TYPE UDT 31
VERSION : 0.0
  STRUCT
   A_FD_OR : BYTE ;	//Feedrate override
   A_DriveEnable : BOOL ;	//Drive test movement enable
   A_AckFixedStop : BOOL ;	//Acknowledge fixed stop reached
   A_SensorFixedStop : BOOL ;	//Sensor fixed stop
   A_ASpDisable : BOOL ;	//Axis/spindle disable
   A_Follow_upMode : BOOL ;	//Follow-up mode
   A_PosMeas1 : BOOL ;	//Position measuring system 1
   A_PosMeas2 : BOOL ;	//Position measuring system 2
   A_ORactive : BOOL ;	//Override active
   A_SWCam : BOOL ;	//SW cam activation
   A_ContrEnable : BOOL ;	//Controller enable
   A_DelDTGSpReset : BOOL ;	//Delete distance to go/Spindle-Reset
   A_Clamp : BOOL ;	//Clamping in progress
   A_RefVal1 : BOOL ;	//Reference point value 1
   A_RefVal2 : BOOL ;	//Reference point value 2
   A_RefVal3 : BOOL ;	//Reference point value 3
   A_RefVal4 : BOOL ;	//Reference point value 4
   A_ExtZO : BOOL ;	//Import external ZO
   A_EnabTravFixedStop : BOOL ;	//Enable travel to fixed stop
   A_FixedFD1 : BOOL ;	//Activate fixed feed 1
   A_FixedFD2 : BOOL ;	//Activate fixed feed 2
   A_FixedFD3 : BOOL ;	//Activate fixed feed 3
   A_FixedFD4 : BOOL ;	//Activate fixed feed 4
   A_VelocSpeedLimit : BOOL ;	//Velocity/spindle speed limitation
   A_PrgtestAxRel : BOOL ;	// Program test axis/spindle release
   A_HW1 : BOOL ;	//Activate handwheel 1
   A_HW2 : BOOL ;	//Activate handwheel 2
   A_HW3 : BOOL ;	//Activate handwheel 3
   A_FDSpStop : BOOL ;	//Feed stop/spindle stop
   A_Disable : BOOL ;	//Traversing key disable
   A_RapidTrOR : BOOL ;	//Rapid traverse override
   A_Minus : BOOL ;	//Traversing key minus
   A_Plus : BOOL ;	//Traversing key plus
   A_INC1 : BOOL ;	//INC1
   A_INC10 : BOOL ;	//INC10
   A_INC100 : BOOL ;	//INC100
   A_INC1000 : BOOL ;	//INC1000
   A_INC10000 : BOOL ;	//INC10000
   A_INCVar : BOOL ;	//INC variable
   A_OEMAxis : BYTE ;	//OEM axis signals
   f7 : BYTE ;
   A_NCASpChanA : BOOL ;	//Assign NC axis/spindle channel A
   A_NCASpChanB : BOOL ;	//Assign NC axis/spindle channel B
   A_NCASpChanC : BOOL ;	//Assign NC axis/spindle channel C
   A_NCASpChanD : BOOL ;	//Assign NC axis/spindle channel D
   A_NCASpStrobe : BOOL ;	//Activation of assignment with pos. edge
   f8_5 : BOOL ;
   f8_6 : BOOL ;
   A_PLCASp : BOOL ;	//Request PLC axis/spindle
   A_Para_A : BOOL ;	//Parameter block servo A
   A_Para_B : BOOL ;	//Parameter block servo B
   A_Para_C : BOOL ;	//Parameter block servo C
   A_LockParSetDef : BOOL ;	//Lock parameter set definition from NC
   f9_4 : BOOL ;
   f9_5 : BOOL ;
   f9_6 : BOOL ;
   f9_7 : BOOL ;
   A_REPOSDelay : BOOL ;	//REPOS DELAY
   f10_1 : BOOL ;
   f10_2 : BOOL ;
   f10_3 : BOOL ;
   f10_4 : BOOL ;
   f10_5 : BOOL ;
   f10_6 : BOOL ;
   f10_7 : BOOL ;
   A_StartBrakeTest : BOOL ;	// Start brake test
   f11_1 : BOOL ;
   f11_2 : BOOL ;
   f11_3 : BOOL ;
   f11_4 : BOOL ;
   f11_5 : BOOL ;
   f11_6 : BOOL ;
   f11_7 : BOOL ;
   A_HWLimitMinus : BOOL ;	//Hardware limit switch minus
   A_HWLimitPlus : BOOL ;	//Hardware limit switch plus
   A_SWLimit2Minus : BOOL ;	//2nd software limit switch minus
   A_SWLimit2Plus : BOOL ;	//2nd software limit switch plus
   A_ModuloLimitEn : BOOL ;	// Modulo limit enabled
   f12_5 : BOOL ;
   f12_6 : BOOL ;
   A_DelayRef : BOOL ;	//Delay reference point approach
   f13 : BYTE ;
   f14 : INT ;
   A_ActGearA : BOOL ;	//Actual gear stage A
   A_ActGearB : BOOL ;	//Actual gear stage B
   A_ActGearC : BOOL ;	//Actual gear stage C
   A_GearChangeOv : BOOL ;	//Gear has changed over
   A_Sp1Syn : BOOL ;	//Re-synchronize spindle 1
   A_Sp2Syn : BOOL ;	//Re-synchronize spindle 2
   A_NoMonitorGear : BOOL ;	//No monitoring when changing gear
   A_DeleteS : BOOL ;	//Delete S value
   A_FD_ORSp : BOOL ;	//Feedrate override for spindle valid
   f17_1 : BOOL ;
   f17_2 : BOOL ;
   f17_3 : BOOL ;
   A_Sp1SynP : BOOL ;	//Re-synchronize spindle 1 f. positioning
   A_Sp2SynP : BOOL ;	//Re-synchronize spindle 2 f. positioning
   A_M3M4Inv : BOOL ;	//Invert M3/M4
   f17_7 : BOOL ;
   f18_0 : BOOL ;
   f18_1 : BOOL ;
   f18_2 : BOOL ;
   f18_3 : BOOL ;
   A_OscilPLC : BOOL ;	//Oscillation via PLC
   A_OscilSpeed : BOOL ;	//enable Oscillation
   A_SetRotDirectRight : BOOL ;	//Setpoint osci. direct. right
   A_SetRotDirectLeft : BOOL ;	//Setpoint osci. direct. left
   A_SpOR : BYTE ;	//Spindle override
   A_UFSwOv : BOOL ;	//Run-up switchover U/F operation
   A_RUEncQuStop : BOOL ;	//Run-up encoder quick stop
   A_Tlimit2 : BOOL ;	//Torque limit 2
   A_SpeedSetpSmooth : BOOL ;	//Speed setpoint smoothing
   f20_4 : BOOL ;
   A_HoldBrakeToOpen : BOOL ;	// holding brake open
   f20_6 : BOOL ;
   f20_7 : BOOL ;
   A_ParA : BOOL ;	//Parameter set selection A
   A_ParB : BOOL ;	//Parameter set selection B
   A_ParC : BOOL ;	//Parameter set selection C
   A_MotA : BOOL ;	//Motor selection A
   A_MotB : BOOL ;	//Motor selection B
   A_MotOK : BOOL ;	//Motor selected
   A_IntegratDisable : BOOL ;	//n controller integrator disable
   A_PulseEnable : BOOL ;	//Pulse enable
   A_SG_SBH : BOOL ;	//Deselection SG/SBH
   A_SBH : BOOL ;	//Deselection of safe standstill
   f22_2 : BOOL ;
   A_SGselect0 : BOOL ;	//Selection SG bit 0
   A_SGselect1 : BOOL ;	//Selection SG bit 1
   f22_5 : BOOL ;
   f22_6 : BOOL ;
   f22_7 : BOOL ;
   A_Transmiss0 : BOOL ;	//Selection Transmission bit 0
   A_Transmiss1 : BOOL ;	//Selection Transmission bit 1
   A_Transmiss2 : BOOL ;	//Selection Transmission bit 2
   f23_3 : BOOL ;
   A_SE : BOOL ;	//Selection SE
   A_BrakeToClose : BOOL ;	// Sinamics: Brake to close
   f23_6 : BOOL ;
   A_TestStop : BOOL ;	//Activate test stop
   A_RotationMonit : BOOL ;	// Stepper motor: Rotation monitoring
   A_ControlAx : BOOL ;	// Control Axis
   f24_2 : BOOL ;
   f24_3 : BOOL ;
   A_TorqComp : BOOL ;	// Torque compensation
   A_ChangSetpOutAss0 : BOOL ;	// Bit value for CTRLOUT_changed - Change setpoint output assignment
   A_ChangSetpOutAss1 : BOOL ;	// Bit value for CTRLOUT_changed - Change setpoint output assignment
   A_MS : BOOL ;	//Master / Slave On
   f25 : BYTE ;
   f26_0 : BOOL ;
   f26_1 : BOOL ;
   f26_2 : BOOL ;
   A_CompContr : BOOL ;	//Compensation controller On
   A_FollowAxOv : BOOL ;	//Enable following axis override
   f26_5 : BOOL ;
   f26_6 : BOOL ;
   f26_7 : BOOL ;
   A_DEPMCS : BOOL ;	// Resume: DEPMCS
   A_DEPBCS : BOOL ;	// Resume: DEPBCS
   A_Corr : BOOL ;	// Resume: Corr
   A_HIAxMove : BOOL ;	// Resume: HIAxMove
   A_StopDEPMCS : BOOL ;	// Stop: DEPMCS
   A_StopDEPBCS : BOOL ;	// Stop: DEPBCS
   A_StopCorr : BOOL ;	// Stop: Corr
   A_StopHIAxMove : BOOL ;	// Stop: HIAxMove
   A_OscillAxExtRev : BOOL ;	// OscillAxExtReversal
   A_AxReset : BOOL ;	// AXRESET
   A_AxResume : BOOL ;	// AXRESUME
   A_SetRP : BOOL ;	//Set reversal point
   A_ChangeRP : BOOL ;	//Change reversal point
   A_StopRP : BOOL ;	//Stop at next reversal point
   A_Stop : BOOL ;	//Stop
   A_PLCAxis : BOOL ;	//PLC checks axis
   f29_0 : BOOL ;
   f29_1 : BOOL ;
   f29_2 : BOOL ;
   f29_3 : BOOL ;
   A_StartGantSynRun : BOOL ;	//Start gantry synchronization run
   A_NoAutoSync : BOOL ;	//No auto sync
   f29_6 : BOOL ;
   f29_7 : BOOL ;
   A_StopSpindle : BOOL ;	//Stop spindle
   A_StartCW : BOOL ;	//Start spindle Clockwise
   A_StartCCW : BOOL ;	//Start spindle Counterclockwise
   A_AutoGearStep : BOOL ;	//Autom. gear step change
   A_PosSpindle : BOOL ;	//Position spindle
   f30_5 : BOOL ;
   f30_6 : BOOL ;
   f30_7 : BOOL ;
   f31_0 : BOOL ;
   f31_1 : BOOL ;
   f31_2 : BOOL ;
   f31_3 : BOOL ;
   A_Resynchronize : BOOL ;	// Resynchronize
   A_DisSync : BOOL ;	// Disable synchronization
   A_Tracksync : BOOL ;	// Track synchronism
   f31_7 : BOOL ;
   f32_0 : BOOL ;
   f32_1 : BOOL ;
   A_extStopA : BOOL ;	//Deselection external Stop A
   A_extStopC : BOOL ;	//Deselection external Stop C
   A_extStopD : BOOL ;	//Deselection external Stop D
   A_extStopE : BOOL ;	//Deselection external Stop E
   f32_6 : BOOL ;
   f32_7 : BOOL ;
   f33_0 : BOOL ;
   f33_1 : BOOL ;
   f33_2 : BOOL ;
   f33_3 : BOOL ;
   A_SGcorr_0 : BOOL ;	//Selection SG-correction Bit 0
   A_SGcorr_1 : BOOL ;	//Selection SG-correction Bit 1
   A_SGcorr_2 : BOOL ;	//Selection SG-correction Bit 2
   A_SGcorr_3 : BOOL ;	//Selection SG-correction Bit 3
   f34 : ARRAY  [34 .. 55 ] OF BYTE ;
   A_FeedDriveCAxEng : BOOL ;	// Seperate feed drive as C axis engaged
   A_SpSpeedDisp : BOOL ;	// Spindle speed display
   A_SpInsideClamp : BOOL ;	// Spindle inside clamping
   f56_3 : BOOL ;
   f56_4 : BOOL ;
   f56_5 : BOOL ;
   f56_6 : BOOL ;
   f56_7 : BOOL ;
   f57 : BYTE ;
   f58 : WORD ;	// FC18: internal
   E_SpNA : BOOL ;	//Spindle/no axis
   E_NCU_Link : BOOL ;	//NCU_link active axis
   E_EncodFreq1 : BOOL ;	//Encoder limit frequency 1 exceeded
   E_EncodFreq2 : BOOL ;	//Encoder limit frequency 2 exceeded
   E_RefSyn1 : BOOL ;	//Referenced/synchronized 1
   E_RefSyn2 : BOOL ;	//Referenced/synchronized 2
   E_ExactCoarse : BOOL ;	//Position reached with exact stop coarse
   E_ExactFine : BOOL ;	//Position reached with exact stop fine
   E_TravRequ : BOOL ;	//Travel request
   E_AxialAlarm : BOOL ;	// Axial alarm
   E_AxisReady : BOOL ;	//Axis ready
   E_Follow_upMode : BOOL ;	//Follow-up mode active
   E_Stat : BOOL ;	//Axis/spindle stationary (n<nmin)
   E_PositContr : BOOL ;	//Position controller active
   E_SpeedContr : BOOL ;	//Speed controller active
   E_CurrentContr : BOOL ;	//Current controller active
   E_SWCam : BOOL ;	//Software cams active
   E_HWOverlay : BOOL ;	//Handwheel overlay active
   E_RevFD : BOOL ;	//Revolutional feedrate active
   E_MeasAct : BOOL ;	//Measuring active
   E_ActTravFStop : BOOL ;	//Activate travel to fixed stop
   E_FixedStop : BOOL ;	//Fixed stop reached
   E_ForceFixedStop : BOOL ;	// Force fixed stop limited
   E_AxContainerRot : BOOL ;	// Axis container rotation active
   E_AxReset : BOOL ;	// Axis reset done
   E_PLCCtrlAx : BOOL ;	// PLCcontrolled axis
   E_AxStop : BOOL ;	// Axis stop active
   E_AxSpDisable : BOOL ;	// Axis/spindle disable active
   E_StopDEPMCS : BOOL ;	// stop DEPMCS active
   E_StopDEPBCS : BOOL ;	// stop DEPBCS active
   E_StopCorr : BOOL ;	// stop Corr active
   E_StopHIAxMove : BOOL ;	// Stop HIAxMove active
   E_HW1 : BOOL ;	//Handwheel 1 active
   E_HW2 : BOOL ;	//Handwheel 2 active
   E_HW3 : BOOL ;	//Handwheel 3 active
   f64_3 : BOOL ;
   E_TReqMinus : BOOL ;	// Travel request minus
   E_TReqPlus : BOOL ;	// Travel request plus
   E_TCMinus : BOOL ;	//Traverse command minus
   E_TCPlus : BOOL ;	//Traverse command plus
   E_INC1 : BOOL ;	//INC1
   E_INC10 : BOOL ;	//INC10
   E_INC100 : BOOL ;	//INC100
   E_INC1000 : BOOL ;	//INC1000
   E_INC10000 : BOOL ;	//INC10000
   E_INCVar : BOOL ;	//INC variable
   f65_6 : BOOL ;
   f65_7 : BOOL ;
   E_OEMAxis : BYTE ;	//OEM axis signals
   f67 : BYTE ;
   E_NCASpChanA : BOOL ;	//NC axis/spindle in channel A
   E_NCASpChanB : BOOL ;	//NC axis/spindle in channel B
   E_NCASpChanC : BOOL ;	//NC axis/spindle in channel C
   E_NCASpChanD : BOOL ;	//NC axis/spindle in channel D
   E_PLCType : BOOL ;	//New type requested by PLC
   E_ChPoss : BOOL ;	//Change axis possible
   E_NeutrASp : BOOL ;	//Neutral axis/spindle
   E_PLCASp : BOOL ;	//PLC axis/spindle
   E_ParS_A : BOOL ;	//Parameter block servo A
   E_ParS_B : BOOL ;	//Parameter block servo B
   E_ParS_C : BOOL ;	//Parameter block servo C
   E_ReposSh : BOOL ;	// Repos shift
   E_ReposShValid : BOOL ;	// Repos shift valid
   E_ReposDelayQuit : BOOL ;	// Repos delay quit
   f70_3 : BOOL ;
   f70_4 : BOOL ;
   f70_5 : BOOL ;
   f70_6 : BOOL ;
   f70_7 : BOOL ;
   E_BrakeTest : BOOL ;	// Brake test active
   f71_1 : BOOL ;
   f71_2 : BOOL ;
   f71_3 : BOOL ;
   f71_4 : BOOL ;
   f71_5 : BOOL ;
   f71_6 : BOOL ;
   E_PLCAxDedic : BOOL ;	// PLC Axis dedicated
   E_MMC_REPOSDelay : BOOL ;	//MMC REPOS DELAY
   f72_1 : BOOL ;
   f72_2 : BOOL ;
   f72_3 : BOOL ;
   f72_4 : BOOL ;
   f72_5 : BOOL ;
   f72_6 : BOOL ;
   f72_7 : BOOL ;
   f73 : BYTE ;
   f74_0 : BOOL ;
   f74_1 : BOOL ;
   f74_2 : BOOL ;
   f74_3 : BOOL ;
   E_ModLimEnAct : BOOL ;	// Modulo limit enabled active
   f74_5 : BOOL ;
   f74_6 : BOOL ;
   f74_7 : BOOL ;
   f75 : BYTE ;
   E_ScratchPulse : BOOL ;	//Scratch pulse
   f76_1 : BOOL ;
   f76_2 : BOOL ;
   f76_3 : BOOL ;
   E_PathAxis : BOOL ;	// Path axis
   E_PosAxis : BOOL ;	//Positioning axis
   E_IndexAxisPos : BOOL ;	//Indexing axis in position
   E_CurvePos : BOOL ;	//Curve axis in position
   E_CollCheckRedSpeed : BOOL ;	//reduced speed of Collisions Check
   f77_1 : BOOL ;
   f77_2 : BOOL ;
   f77_3 : BOOL ;
   f77_4 : BOOL ;
   f77_5 : BOOL ;
   f77_6 : BOOL ;
   f77_7 : BOOL ;
   E_FPosAxis : REAL ;	//F function (REAL format) for positioning axes
   E_SetpGearA : BOOL ;	//Setpoint gear stage A
   E_SetpGearB : BOOL ;	//Setpoint gear stage B
   E_SetpGearC : BOOL ;	//Setpoint gear stage C
   E_GearChange : BOOL ;	//Gear changeover
   f82_4 : BOOL ;
   f82_5 : BOOL ;
   f82_6 : BOOL ;
   f82_7 : BOOL ;
   E_SpeedLimit : BOOL ;	//Speed limit exceeded
   E_SetSpeedLimit : BOOL ;	//Setpoint speed limited
   E_SetSpeedIncreased : BOOL ;	//Setpoint speed increased
   E_GeoMonit : BOOL ;	//Geometry monitoring
   E_SupportAreaViol : BOOL ;	//Support area limits violated
   E_SetRange : BOOL ;	//Spindle in setpoint range
   E_SpeedMonit : BOOL ;	//Speed monitoring
   E_ActRotRight : BOOL ;	//Actual rotation direction right
   E_ConstCuttSpeed : BOOL ;	//Const. cutting speed active
   E_SUG : BOOL ;	//SUG active (grinding wheel surface speed)
   E_CLG : BOOL ;	//CLG active
   E_Tapping : BOOL ;	//Tapping without compensating chuck
   E_SyncMode : BOOL ;	//Synchronous mode spindle active
   E_PosMode : BOOL ;	//Positioning mode spindle active
   E_OscillMode : BOOL ;	//Oscillation mode spindle active
   E_ContrMode : BOOL ;	//Control mode spindle active
   f85_0 : BOOL ;
   f85_1 : BOOL ;
   f85_2 : BOOL ;
   f85_3 : BOOL ;
   f85_4 : BOOL ;
   E_SpInPosition : BOOL ;	// Spindle in position
   f85_6 : BOOL ;
   f85_7 : BOOL ;
   E_MFunct : INT ;	//M function (INT) for spindle
   E_SFunct : REAL ;	//S function (REAL) for spindle
   E_SetUpMode : BOOL ;	//Set-up mode active
   E_RUEncDisabl : BOOL ;	//Run-up encoder disable active
   E_Tlimit2 : BOOL ;	//Torque limit 2 active
   E_SpeedSetpSmooth : BOOL ;	//Speed setpoint smoothing active
   E_RLIact : BOOL ;	// RLI active
   E_HoldBrakeOpened : BOOL ;	// holding brake opened
   E_EarthFaultDetec : BOOL ;	// earth-fault detection
   f92_7 : BOOL ;
   E_ParA : BOOL ;	//Active parameter set A
   E_ParB : BOOL ;	//Active parameter set B
   E_ParC : BOOL ;	//Active parameter set C
   E_MotA : BOOL ;	//Active motor A
   E_MotB : BOOL ;	//Active motor B
   E_MotOK : BOOL ;	//Drive ready
   E_IntegratDisable : BOOL ;	//n controller integrator disabled
   E_PulseEnable : BOOL ;	//Pulses enabled
   E_MTempWarn : BOOL ;	//Temperature prewarning motor
   E_HTempWarn : BOOL ;	//Temperature prewarning heat sink
   E_RUComplete : BOOL ;	//Ramp-up complete
   E_MdMdx : BOOL ;	//Md<Mdx
   E_NactNmin : BOOL ;	//nact<nmin
   E_NactNx : BOOL ;	//nact<nx
   E_NactNset : BOOL ;	//nact<nset
   E_Message : BOOL ;	//Variable message function
   E_UDClessAlThreshold : BOOL ;	//UDC-link < alarm threshold
   E_RetractVolt : BOOL ;	// Fall short of retract voltage
   E_Generator : BOOL ;	// Generator active
   E_MinGeneratorVolt : BOOL ;	// Fall short of min. generator voltage
   E_SpeedThreshold : BOOL ;	// Speed threshold star/delta
   f95_5 : BOOL ;
   f95_6 : BOOL ;
   E_PowerSecI2TLimit : BOOL ;	// Power Section I2T limit
   E_SpindleMonit : BOOL ;	//Error spindle monitoring
   E_AxisCtrl : BOOL ;	// Axis control active
   E_MSFine : BOOL ;	// Master/Slave fine
   E_MSCoarse : BOOL ;	// Master/Slave coarse
   E_MSCompContr : BOOL ;	// Master/Slave Compensation controller activ
   E_BitValCtrlOutChang0 : BOOL ;	// Bit value for CTRLOUT_changed 0:  Change setpoint output assignment
   E_BitValCtrlOutChang1 : BOOL ;	// Bit value for CTRLOUT_changed 1:  Change setpoint output assignment
   E_MS : BOOL ;	//Master/ slave active
   f97 : BYTE ;
   E_SyncronFine : BOOL ;	//Synchronism fine
   E_SyncronCoarse : BOOL ;	//Synchronism coarse
   E_ActValCoupling : BOOL ;	//Actual value coupling
   f98_3 : BOOL ;
   E_OverlayMotion : BOOL ;	//Overlaid motion
   E_SWL : BOOL ;	//Speed warning limit reached
   E_AWL : BOOL ;	//Acceleration warning limit reached
   E_EmRetr : BOOL ;	//Emergency retraction active
   E_MasterSp : BOOL ;	//Master spindle
   E_SlaveSp : BOOL ;	//Slave spindle
   f99_2 : BOOL ;
   E_AxisAccel : BOOL ;	//Axis accelerated
   E_Sync : BOOL ;	//Synchronization active
   E_MSR : BOOL ;	//Max speed reached
   E_MAR : BOOL ;	//Max acceleration reached
   E_EmRetrEnabl : BOOL ;	//Emergency retraction enabled
   f100_0 : BOOL ;
   f100_1 : BOOL ;
   E_OscillAxExtRev : BOOL ;	// OscillAxExt Reversal active
   E_StopOscill : BOOL ;	//Oscillation cannot start
   E_ErrorOscill : BOOL ;	//Error during oscillation
   E_SparkOut : BOOL ;	//Spark-out active
   E_OscillMotion : BOOL ;	//Oscillation motion active
   E_Oscill : BOOL ;	//Oscillation active
   f101_0 : BOOL ;
   f101_1 : BOOL ;
   E_GantCOLimit : BOOL ;	//Gantry cut-off limit exceeded
   E_GantWarn : BOOL ;	//Gantry warning limit exceeded
   E_SynRunStart : BOOL ;	//Synchronization run ready to start
   E_GantGroupSyn : BOOL ;	//Gantry grouping is synchronous
   E_GantLeadAxis : BOOL ;	//Gantry leading axis
   E_GantAxis : BOOL ;	//Gantry axis
   f102 : INT ;
   E_AIAxis : ARRAY  [1 .. 31 ] OF BOOL ;	//Active infeed axis[1..31]
   E_SG_SBH : BOOL ;	//Active SG/SBH
   E_ErrLifeS_CRC : BOOL ;	// Error lifesign or CRC-error
   E_ImpdelNCK : BOOL ;	//Delete pulses NCK
   r108_3 : BOOL ;
   r108_4 : BOOL ;
   r108_5 : BOOL ;
   E_SE2 : BOOL ;	//SE 2 active
   E_SRef : BOOL ;	//Axis safely referenced
   E_SN1Plus : BOOL ;	//Actual position > cam position SN1+
   E_SN1Minus : BOOL ;	//Actual position > cam position SN1-
   E_SN2Plus : BOOL ;	//Actual position > cam position SN2+
   E_SN2Minus : BOOL ;	//Actual position > cam position SN2-
   E_SN3Plus : BOOL ;	//Actual position > cam position SN3+
   E_SN3Minus : BOOL ;	//Actual position > cam position SN3-
   E_SN4Plus : BOOL ;	//Actual position > cam position SN4+
   E_SN4Minus : BOOL ;	//Actual position > cam position SN4-
   f110_0 : BOOL ;
   E_SBH : BOOL ;	//Active SBH
   f110_2 : BOOL ;
   E_SG_0 : BOOL ;	//Active SG 0
   E_SG_1 : BOOL ;	//Active SG 1
   E_n_nx : BOOL ;	//n < nx
   f110_6 : BOOL ;
   f110_7 : BOOL ;
   f111_0 : BOOL ;
   f111_1 : BOOL ;
   f111_2 : BOOL ;
   f111_3 : BOOL ;
   E_StopAB : BOOL ;	//Stop A/B active
   E_StopC : BOOL ;	//Stop C active
   E_StopD : BOOL ;	//Stop D active
   E_StopE : BOOL ;	//Stop E active
   E_CamRangeTr1 : BYTE ;	//Cam Range for Cam Track 1
   E_CamRangeTr2 : BYTE ;	//Cam Range for Cam Track 2
   E_CamRangeTr3 : BYTE ;	//Cam Range for Cam Track 3
   E_CamRangeTr4 : BYTE ;	//Cam Range for Cam Track 4
   f116 : BYTE ;
   E_CamTrack1 : BOOL ;	//Cam Track 1
   E_CamTrack2 : BOOL ;	//Cam Track 2
   E_CamTrack3 : BOOL ;	//Cam Track 3
   E_CamTrack4 : BOOL ;	//Cam Track 4
   f117_4 : BOOL ;
   f117_5 : BOOL ;
   f117_6 : BOOL ;
   f117_7 : BOOL ;
   E_CamRangeBitTr1 : ARRAY  [0 .. 14 ] OF //Cam Range Bits for Cam Track 1
   BOOL ;
   E_CamRangeBitTr2 : ARRAY  [0 .. 14 ] OF //Cam Range Bits for Cam Track 2
   BOOL ;
   E_CamRangeBitTr3 : ARRAY  [0 .. 14 ] OF //Cam Range Bits for Cam Track 3
   BOOL ;
   E_CamRangeBitTr4 : ARRAY  [0 .. 14 ] OF //Cam Range Bits for Cam Track 4
   BOOL ;
  END_STRUCT ;	
END_TYPE

TYPE UDT 71
VERSION : 0.0
  STRUCT
   IFNo : ARRAY  [1 .. 16 ] OF BOOL ;	//Interface [no.] active
   Quit : ARRAY  [1 .. 16 ] OF BOOL ;	//perform Quit-End
   IF : ARRAY  [1 .. 16 ] OF STRUCT
    Loading : BOOL ;
    Unloading : BOOL ;
    Reloading : BOOL ;
    Positioning : BOOL ;
    PosbyProgram : BOOL ;	//Positioning by CNC Program with POSM
    f0_5 : BOOL ;
    f0_6 : BOOL ;
    f0_7 : BOOL ;
    PerfStatusError : BOOL ;
    Channel : BYTE ;	//Assigned channel
    TMno : BYTE ;	//Tool management no.
    Free1 : DINT ;	//Unassigned parameter 1
    Free2 : DINT ;	//Unassigned parameter 2
    Free3 : DINT ;	//Unassigned parameter 3
    IdentLoad : INT ;	//Identification for loading/unloading station
    NoLoad : INT ;	//No. of loading station
    SMag : INT ;	//Magazine no. (source) for unloading/reloading/pos.
    SLoc : INT ;	//Location no. (source) for unloading/reloading/pos.
    TMag : INT ;	//Magazine no. (target) for loading/reloading
    TLoc : INT ;	//Location no. (target) for loading/reloading
    WithoutMagMoving : BOOL ;	//HMI Data: Without Magazine Moving
    Res2 : BYTE ;
   END_STRUCT ;
  END_STRUCT ;	
END_TYPE

TYPE UDT 72
VERSION : 0.0
  STRUCT
   IFNo : ARRAY  [1 .. 16 ] OF BOOL ;	//Interface [no.] active
   Quit : ARRAY  [1 .. 16 ] OF BOOL ;	//perform Quit-End
   IF : ARRAY  [1 .. 16 ] OF STRUCT
    Comp : BOOL ;	//Compulsory change
    Perform : BOOL ;	//Perform change
    Prepare : BOOL ;	//Prepare change
    T0 : BOOL ;	//T0 programmed
    OldTinDBW42 : BOOL ;	//ZWS No. of Old Tool in DBW (n+42)
    ManTIn : BOOL ;	//Put in Tool in Spindle manual
    ManTOut : BOOL ;	//Get out Tool from Spindle manual
    SpiTRSpi : BOOL ;	//Spindle Tool remains in spindle
    PerfStatusError : BOOL ;
    Channel : BYTE ;	//Assigned channel
    TMno : BYTE ;	//Tool management no.
    Free1 : DINT ;	//Unassigned parameter 1
    Free2 : DINT ;	//Unassigned parameter 2
    Free3 : DINT ;	//Unassigned parameter 3
    IdentBuff : INT ;	//Buffer identification (fixed value 9998)
    NoBuff : INT ;	//Relative location (target) in the buffer
    SMag : INT ;	//Magazine no. (source) for new tool
    SLoc : INT ;	//Location no. (source) for new tool
    TMag : INT ;	//Magazine no. (target) for old tool
    TLoc : INT ;	//Location no. (target) for old tool
    LocType : INT ;	//Tool new: location type
    SLeft : INT ;	//Tool new: size left
    SRight : INT ;	//Tool new: size right
    STop : INT ;	//Tool new: size top
    SBottom : INT ;	//Tool new: size bottom
    ActTool : BOOL ;	//Active tool
    ToolEnabl : BOOL ;	//Tool enabled
    ToolDisab : BOOL ;	//Tool disabled
    Measured : BOOL ;	//Tool measured
    Prewarn : BOOL ;	//Prewarning limit reached
    ToolChange : BOOL ;	//Tool being changed
    FixedLoc : BOOL ;	//Tool fixed location coded
    ToolUsed : BOOL ;	//Tool was in use
    ToolInBuff : BOOL ;	//ID for tools in buffer
    IgnoreDisab : BOOL ;	//Ignore disabled
    TBUnloaded : BOOL ;	//To be unloaded
    TBLoaded : BOOL ;	//To be loaded
    MasterTool : BOOL ;	//Master tool
    n39_5 : BOOL ;	//reserved
    n39_6 : BOOL ;	//reserved
    n39_7 : BOOL ;	//reserved
    T_no : INT ;	//Tool new: T no.
    OldTZWSNo : INT ;	//ZWS No. of Old Tool
    MyMag : INT ;
    MyPlace : INT ;
   END_STRUCT ;
  END_STRUCT ;	
END_TYPE

TYPE UDT 73
VERSION : 0.0
  STRUCT
   IfNo : ARRAY  [1 .. 16 ] OF BOOL ;	//Interface [no.] active
   Quit : ARRAY  [1 .. 16 ] OF BOOL ;	//perform Quit-End
   IF : ARRAY  [1 .. 16 ] OF STRUCT
    Comp : BOOL ;	//Compulsory change
    Perform : BOOL ;	//Perform change
    f0_2 : BOOL ;
    T0 : BOOL ;	//T0 programmed
    f0_4 : BOOL ;
    f0_5 : BOOL ;
    ManTOut : BOOL ;	//Get out Tool from Holder manual
    f0_7 : BOOL ;
    PerfStatusError : BOOL ;
    Channel : BYTE ;	//Assigned channel
    TMno : BYTE ;	//Tool management no.
    Free1 : DINT ;	//Unassigned parameter 1
    Free2 : DINT ;	//Unassigned parameter 2
    Free3 : DINT ;	//Unassigned parameter 3
    KennZWS : INT ;	//Reserved (buffer identification)
    NoBuff : INT ;	//Rel. location in buffer (res.)
    SMag : INT ;	//Magazine no. of turret
    SLoc : INT ;	//Location no. for new tool
    TMag : INT ;	//Magazine no. of turret (res.)
    TLoc : INT ;	//Location no. for old tool
    LocType : INT ;	//Tool new: location type
    SLeft : INT ;	//Tool new: size left
    SRight : INT ;	//Tool new: size right
    STop : INT ;	//Tool new: size top
    SBottom : INT ;	//Tool new: size bottom
    ActTool : BOOL ;	//Active tool
    ToolEnabl : BOOL ;	//Tool enabled
    ToolDisab : BOOL ;	//Tool disabled
    Measured : BOOL ;	//Tool measured
    Prewarn : BOOL ;	//Prewarning limit reached
    ToolChange : BOOL ;	//Tool being changed
    FixedLoc : BOOL ;	//Tool fixed location coded
    ToolUsed : BOOL ;	//Tool was in use
    ToolInBuff : BOOL ;	//ID for tools in buffer
    IgnoreDisab : BOOL ;	//Ignore disabled
    TBUnloaded : BOOL ;	//To be unloaded
    TBLoaded : BOOL ;	//To be loaded
    MasterTool : BOOL ;	//Master tool
    n39_5 : BOOL ;	//reserved
    n39_6 : BOOL ;	//reserved
    n39_7 : BOOL ;	//reserved
    T_no : INT ;	//Tool new: T no.
    MyPlace : INT ;
   END_STRUCT ;
  END_STRUCT ;	
END_TYPE

TYPE UDT 77
VERSION : 0.0
  STRUCT
   MCP1In : ARRAY  [0 .. 7 ] OF BYTE ;
   MCP1Out : ARRAY  [0 .. 7 ] OF BYTE ;
   MCP1StatSend : DWORD ;
   MCP1StatRec : DWORD ;
   MCP2In : ARRAY  [0 .. 7 ] OF BYTE ;
   MCP2Out : ARRAY  [0 .. 7 ] OF BYTE ;
   MCP2StatSend : DWORD ;
   MCP2StatRec : DWORD ;
   BHGIn : ARRAY  [0 .. 5 ] OF BYTE ;
   Filler : ARRAY  [0 .. 5 ] OF BYTE ;
   BHGOut : ARRAY  [0 .. 19 ] OF BYTE ;
   BHGStatSend : DWORD ;
   BHGStatRec : DWORD ;
  END_STRUCT ;	
END_TYPE

TYPE "MM4_Control_Word"	// UDT 91
AUTHOR : PROTEKNO
FAMILY : Profibus
NAME : MM4
VERSION : 0.1
  STRUCT
   Bit_8 : BOOL ;	//1=Jog right on/ 0=Jog right off
   Bit_9 : BOOL ;	//1=Jog left on / 0=Jog left off
   Bit_10 : BOOL ;	//1=Setpoint valid / 0=Setpoint invalid
   Bit_11 : BOOL ;	//1=Setpoint inverted/ 0=Setpoint is not inverted
   Bit_12 : BOOL ;	//-
   Bit_13 : BOOL ;	//1=Motor potentiometer UP / 0=No meaning
   Bit_14 : BOOL ;	//1=Motor potentiometer Down / 0=No meaning
   Bit_15 : BOOL ;	//1=Local control active(BOP/AOP) / 0=Remote control active
   Bit_0 : BOOL ;	//1=On/ 0=OFF
   Bit_1 : BOOL ;	//1=Operating condition/ 0=OFF2 - pulse disable
   Bit_2 : BOOL ;	//1=Operating condition/ 0=OFF3 - Rapid stop
   Bit_3 : BOOL ;	//1=Enable operation/ 0=Disable operation
   Bit_4 : BOOL ;	//1=Operating condition/ 0=Disable RFG
   Bit_5 : BOOL ;	//1=Enable RFG / 0=Stop RFG
   Bit_6 : BOOL ;	//1=Enable setpoint/ 0=Disable setpoint
   Bit_7 : BOOL ;	//1=fault acknowledge / 0=No meaning
  END_STRUCT ;	
END_TYPE

TYPE "MM4_Status_Word"	// UDT 92
AUTHOR : PROTEKNO
FAMILY : Profibus
NAME : MM4
VERSION : 0.1
  STRUCT
   Bit_8 : BOOL ;	//1=No setpoint-act.val. deviation/ 0=setpoint-act.val. deviation
   Bit_9 : BOOL ;	//1=Master control requested/ 0=Local operation
   Bit_10 : BOOL ;	//1=fmax reached/ 0=fmax not reached
   Bit_11 : BOOL ;	//1= / 0=Alarm:Motor at current limit
   Bit_12 : BOOL ;	//1= / 0=Motor holding brake
   Bit_13 : BOOL ;	//1= / 0=Motor overload
   Bit_14 : BOOL ;	//1= CW rotation / 0= CCW rotation
   Bit_15 : BOOL ;	//1= /0=Converter overload
   Bit_0 : BOOL ;	//1=Ready for On/ 0=Not ready for On
   Bit_1 : BOOL ;	//1=Ready for run/  0=Not ready for run
   Bit_2 : BOOL ;	//1=Operation enabled/ 0=Operation disabled
   Bit_3 : BOOL ;	//1=Fault active / 0=No fault active
   Bit_4 : BOOL ;	//1=No OFF2 command applied / 0=OFF2 command applied
   Bit_5 : BOOL ;	//1=No OFF3 command applied / 0=OFF3 command applied
   Bit_6 : BOOL ;	//1=Starting lockout / 0=No Starting lockout
   Bit_7 : BOOL ;	//1=Alarm is active / 0= Alarm is active
  END_STRUCT ;	
END_TYPE

TYPE UDT 1002
VERSION : 0.0
  STRUCT 	//Offset 0
   Chan : ARRAY  [1 .. 10 ] OF STRUCT 	//From Channel 1 to Channel 10
    FDD : ARRAY  [0 .. 15 ] OF //Feed disable
    BOOL ;
    RID : ARRAY  [0 .. 15 ] OF //Read-in disable
    BOOL ;
    NCSD : ARRAY  [0 .. 15 ] OF //NC start disable
    BOOL ;
    FdStop_1 : ARRAY  [0 .. 15 ] OF //Feed stop GEOaxis 1
    BOOL ;
    FdStop_2 : ARRAY  [0 .. 15 ] OF //Feed stop GEOaxis 2
    BOOL ;
    FdStop_3 : ARRAY  [0 .. 15 ] OF //Feed stop GEOaxis 3
    BOOL ;
   END_STRUCT ;	//without Alarmno for Chan (120 Byte)
//Offset 120
   Axis : ARRAY  [1 .. 31 ] OF STRUCT 	//From Axis 1 to Axis 31
    FdStop : ARRAY  [0 .. 15 ] OF //Feed stop axis/spindle 1
    BOOL ;
   END_STRUCT ;	//without Alarmno for Axis (62 Byte)
//Offset 182
   ZInfo0 : ARRAY  [0 .. 63 ] OF WORD ;	//Additional Value for UserAlarms 700000 to 700063
//Offset 310
   ChanA : ARRAY  [1 .. 10 ] OF STRUCT 	//From Channel 1 to Channel 10
    FDD_5C00xx : ARRAY  [0 .. 15 ] OF //Feed disable A.no.51000-510015
    BOOL ;
    FDD_RID_5C01xx : ARRAY  [0 .. 31 ] OF //Feed and read-in disable A.no.510100-510131
    BOOL ;
    RID_5C02xx : ARRAY  [0 .. 31 ] OF //Read-in disable A.no.510200-510231
    BOOL ;
    NCSD_5C03xx : ARRAY  [0 .. 15 ] OF //NC start disable A.no.510300-510315
    BOOL ;
    FdStop_1_5C11xx : ARRAY  [0 .. 15 ] OF //Feed stop GEOaxis 1 A.no.511100-511115
    BOOL ;
    FdStop_2_5C12xx : ARRAY  [0 .. 15 ] OF //Feed stop GEOaxis 2 A.no.511200-511215
    BOOL ;
    FdStop_3_5C13xx : ARRAY  [0 .. 15 ] OF //Feed stop GEOaxis 3 A.no.511300-511315
    BOOL ;
   END_STRUCT ;	//Alarmno for Chan are 5Cxxxx; C is the ChannelNo, except Channel 10. Channel 10
   AxisA : ARRAY  [1 .. 32 ] OF STRUCT 	//From Axis 1 to Axis 31
    AAFdStop60AAxx : ARRAY  [0 .. 15 ] OF //Feed stop axis/spindle
    BOOL ;
   END_STRUCT ;	//Alarmno for Axis are 60AAxx; A is the Axisno.
//Offset 554
   UserA : ARRAY  [0 .. 31 ] OF STRUCT
    A70UUxx : ARRAY  [0 .. 63 ] OF //Alarm 700000-700063 (user area 0)
    BOOL ;
   END_STRUCT ;	//Alarmno for UserAlarms are 7yUUxx; U is the Userarea, y = Db1004.UserDek2No[U]
  END_STRUCT ;	
END_TYPE

// FB 1: know-how protected block, not included

// FB 2: know-how protected block, not included

// FB 3: know-how protected block, not included

// FB 4: know-how protected block, not included

// FB 5: know-how protected block, not included

// FB 7: know-how protected block, not included

// FB 9: know-how protected block, not included

// FB 10: know-how protected block, not included

// FB 11: know-how protected block, not included

// FB 29: know-how protected block, not included

FUNCTION_BLOCK "FB Analogiche"	// FB 200
TITLE = FB Gestione Analogiche
VERSION : 0.1
VAR_INPUT
  IN1 : INT ;
  IN2 : INT ;
  IN3 : INT ;
  IN1_Soglia1_Min : INT ;
  IN1_Soglia1_Max : INT ;
  IN1_Soglia2_Min : INT ;
  IN1_Soglia2_Max : INT ;
  IN2_Soglia1_Min : INT ;
  IN2_Soglia1_Max : INT ;
  IN2_Soglia2_Min : INT ;
  IN2_Soglia2_Max : INT ;
  IN3_Soglia1_Min : INT ;
  IN3_Soglia1_Max : INT ;
  IN3_Soglia2_Min : INT ;
  IN3_Soglia2_Max : INT ;
  Isteresi1 : INT ;
  Isteresi2 : INT ;
  Isteresi3 : INT ;
END_VAR
VAR_OUTPUT
  IN1_Soglia1OK : BOOL ;
  IN1_Soglia2OK : BOOL ;
  IN2_Soglia1OK : BOOL ;
  IN2_Soglia2OK : BOOL ;
  IN3_Soglia1OK : BOOL ;
  IN3_Soglia2OK : BOOL ;
END_VAR
VAR
  Timer1 : SFB 4;
  Timer2 : SFB 4;
  Timer3 : SFB 4;
  Timer4 : SFB 4;
  Timer5 : SFB 4;
  Timer6 : SFB 4;
  Timer7 : SFB 4;
  Timer8 : SFB 4;
END_VAR
VAR_TEMP
  Ret_Val1 : WORD ;
  Ret_Val2 : WORD ;
  Ret_Val3 : WORD ;
  Out1 : REAL ;
  Out2 : REAL ;
  Out3 : REAL ;
  ValoreMin : INT ;
  ValoreMax : INT ;
END_VAR
BEGIN
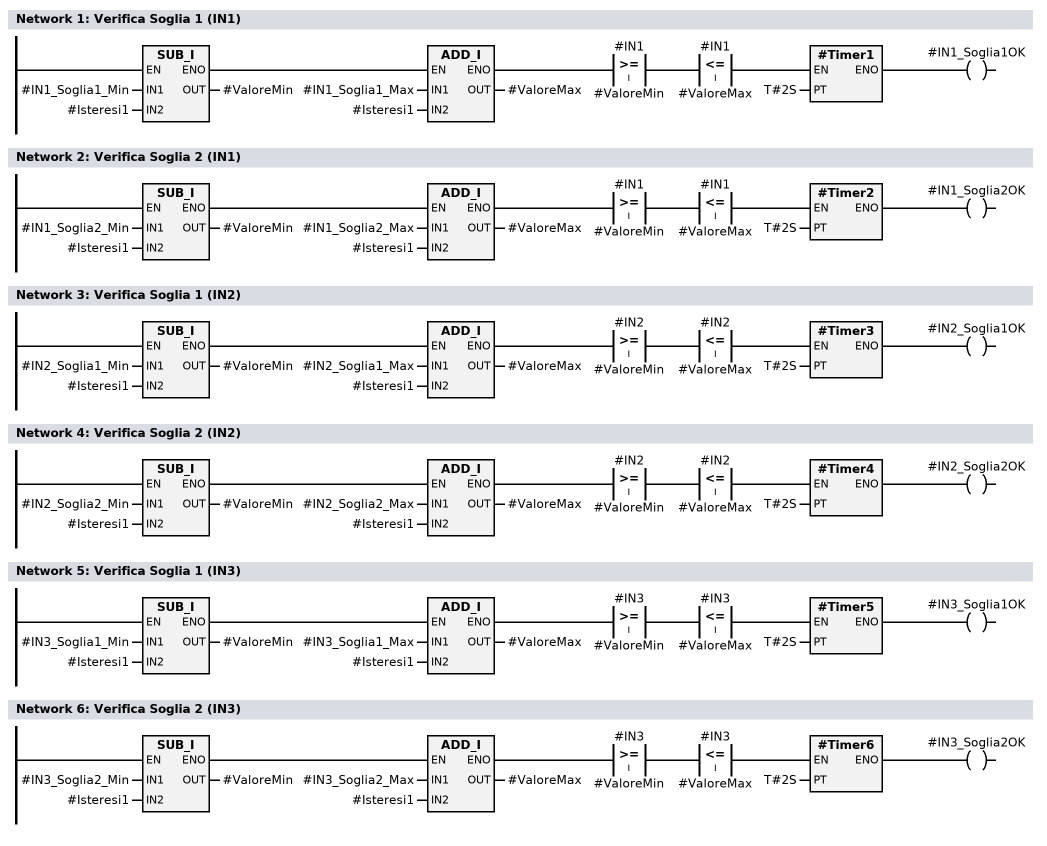
NETWORK
TITLE = Verifica Soglia 1 (IN1)
      A(;
      A(;
      L     #IN1_Soglia1_Min;
      L     #Isteresi1;
      -I;
      T     #ValoreMin;
      AN    OV;
      SAVE;
      CLR;
      A     BR;
      );
      JNB   _001;
      L     #IN1_Soglia1_Max;
      L     #Isteresi1;
      +I;
      T     #ValoreMax;
      AN    OV;
      SAVE;
      CLR;
_001: A     BR;
      );
      A(;
      L     #IN1;
      L     #ValoreMin;
      >=I;
      );
      A(;
      L     #IN1;
      L     #ValoreMax;
      <=I;
      );
      JNB   _002;
      CALL  #Timer1 (
           PT                       := T#2S);
_002: A     BR;
      =     #IN1_Soglia1OK;
NETWORK
TITLE = Verifica Soglia 2 (IN1)
      A(;
      A(;
      L     #IN1_Soglia2_Min;
      L     #Isteresi1;
      -I;
      T     #ValoreMin;
      AN    OV;
      SAVE;
      CLR;
      A     BR;
      );
      JNB   _003;
      L     #IN1_Soglia2_Max;
      L     #Isteresi1;
      +I;
      T     #ValoreMax;
      AN    OV;
      SAVE;
      CLR;
_003: A     BR;
      );
      A(;
      L     #IN1;
      L     #ValoreMin;
      >=I;
      );
      A(;
      L     #IN1;
      L     #ValoreMax;
      <=I;
      );
      JNB   _004;
      CALL  #Timer2 (
           PT                       := T#2S);
_004: A     BR;
      =     #IN1_Soglia2OK;
NETWORK
TITLE = Verifica Soglia 1 (IN2)
      A(;
      A(;
      L     #IN2_Soglia1_Min;
      L     #Isteresi1;
      -I;
      T     #ValoreMin;
      AN    OV;
      SAVE;
      CLR;
      A     BR;
      );
      JNB   _005;
      L     #IN2_Soglia1_Max;
      L     #Isteresi1;
      +I;
      T     #ValoreMax;
      AN    OV;
      SAVE;
      CLR;
_005: A     BR;
      );
      A(;
      L     #IN2;
      L     #ValoreMin;
      >=I;
      );
      A(;
      L     #IN2;
      L     #ValoreMax;
      <=I;
      );
      JNB   _006;
      CALL  #Timer3 (
           PT                       := T#2S);
_006: A     BR;
      =     #IN2_Soglia1OK;
NETWORK
TITLE = Verifica Soglia 2 (IN2)
      A(;
      A(;
      L     #IN2_Soglia2_Min;
      L     #Isteresi1;
      -I;
      T     #ValoreMin;
      AN    OV;
      SAVE;
      CLR;
      A     BR;
      );
      JNB   _007;
      L     #IN2_Soglia2_Max;
      L     #Isteresi1;
      +I;
      T     #ValoreMax;
      AN    OV;
      SAVE;
      CLR;
_007: A     BR;
      );
      A(;
      L     #IN2;
      L     #ValoreMin;
      >=I;
      );
      A(;
      L     #IN2;
      L     #ValoreMax;
      <=I;
      );
      JNB   _008;
      CALL  #Timer4 (
           PT                       := T#2S);
_008: A     BR;
      =     #IN2_Soglia2OK;
NETWORK
TITLE = Verifica Soglia 1 (IN3)
      A(;
      A(;
      L     #IN3_Soglia1_Min;
      L     #Isteresi1;
      -I;
      T     #ValoreMin;
      AN    OV;
      SAVE;
      CLR;
      A     BR;
      );
      JNB   _009;
      L     #IN3_Soglia1_Max;
      L     #Isteresi1;
      +I;
      T     #ValoreMax;
      AN    OV;
      SAVE;
      CLR;
_009: A     BR;
      );
      A(;
      L     #IN3;
      L     #ValoreMin;
      >=I;
      );
      A(;
      L     #IN3;
      L     #ValoreMax;
      <=I;
      );
      JNB   _00a;
      CALL  #Timer5 (
           PT                       := T#2S);
_00a: A     BR;
      =     #IN3_Soglia1OK;
NETWORK
TITLE = Verifica Soglia 2 (IN3)
      A(;
      A(;
      L     #IN3_Soglia2_Min;
      L     #Isteresi1;
      -I;
      T     #ValoreMin;
      AN    OV;
      SAVE;
      CLR;
      A     BR;
      );
      JNB   _00b;
      L     #IN3_Soglia2_Max;
      L     #Isteresi1;
      +I;
      T     #ValoreMax;
      AN    OV;
      SAVE;
      CLR;
_00b: A     BR;
      );
      A(;
      L     #IN3;
      L     #ValoreMin;
      >=I;
      );
      A(;
      L     #IN3;
      L     #ValoreMax;
      <=I;
      );
      JNB   _00c;
      CALL  #Timer6 (
           PT                       := T#2S);
_00c: A     BR;
      =     #IN3_Soglia2OK;
END_FUNCTION_BLOCK

// FC 2: know-how protected block, not included

// FC 3: know-how protected block, not included

// FC 5: know-how protected block, not included

// FC 7: know-how protected block, not included

// FC 8: know-how protected block, not included

// FC 9: know-how protected block, not included

// FC 10: know-how protected block, not included

FUNCTION FC 12 : VOID
AUTHOR : NUMERIK
FAMILY : _800D
NAME : Basics
VERSION : 1.5
VAR_INPUT
  Chan : BYTE ;	//Index of Chan
END_VAR
BEGIN
// (block stored without names or comments; labels and parameter names are numbered)
END_FUNCTION

// FC 13: know-how protected block, not included

// FC 17: know-how protected block, not included

// FC 18: know-how protected block, not included

// FC 19: know-how protected block, not included

// FC 21: know-how protected block, not included

// FC 22: know-how protected block, not included

// FC 24: know-how protected block, not included

// FC 25: know-how protected block, not included

// FC 26: know-how protected block, not included

FUNCTION "Nck-plc" : VOID	// FC 95
VERSION : 0.1
BEGIN
NETWORK
TITLE =
      CALL  "GET" , DB 95 (
           DIW 2                    := 1,
           DIW 4                    := W#16#1002,
           DIW 6                    := 10,
           DIW 8                    := 120,
           DID 10                   := P#DBX 0.0);
END_FUNCTION

FUNCTION "FC Timer" : VOID	// FC 97
TITLE = Setta Timer Esterno
AUTHOR : Asamec
VERSION : 0.0
VAR_INPUT
  VALORE_TEMPO : INT ;
  Base : INT ;	//1=Decimi, 2=Secondi , 3=10*sec
END_VAR
VAR_OUTPUT
  VALORE_PER_TIMER : S5TIME ;	//VALORE DA CARICARE SUL TIMER
END_VAR
VAR_TEMP
  VALORE : DWORD ;
END_VAR
BEGIN
NETWORK
TITLE =
      L     #VALORE_TEMPO;
      ITB;
      L     W#16#FFF;
      AW;
      T     #VALORE;
      L     #Base;
      L     1;
      ==I;
      JC    M001;
      TAK;
      L     2;
      ==I;
      JC    M002;
      TAK;
      L     3;
      ==I;
      JC    M003;
      JU    M004;
M001: NOP   0;	// decimi
      L     W#16#1000;
      L     #VALORE;
      OW;
      T     #VALORE_PER_TIMER;
      JU    M004;
M002: NOP   0;	// secondi
      L     W#16#2000;
      L     #VALORE;
      OW;
      T     #VALORE_PER_TIMER;
      JU    M004;
M003: NOP   0;	// 10*sec
      L     W#16#3000;
      L     #VALORE;
      OW;
      T     #VALORE_PER_TIMER;
M004: NOP   0;
END_FUNCTION

FUNCTION "FC DecodM" : VOID	// FC 98
TITLE = Decodifica Funzioni M
AUTHOR : Asamec
VERSION : 0.0
VAR_INPUT
  VALORE_CODICE_M1 : DINT ;	//PRIMA FUNZIONE M
  VALORE_CODICE_M2 : DINT ;	//SECONDA FUNZIONE M
  VALORE_CODICE_M3 : DINT ;	//TERZA FUNZIONE M
  VALORE_CODICE_M4 : DINT ;	//QUARTA FUNZIONE M
  VALORE_CODICE_M5 : DINT ;	//QUINTA FUNZIONE M
  NR_MAX_DECOD : INT ;	//MASSIMO NUMERO DA DECODIFICARE
END_VAR
VAR_OUTPUT
  M_ATTIVA : BOOL ;	//FUNZIONE M PRESENTE
END_VAR
VAR_TEMP
  COUNT_M1 : DWORD ;
  COUNT_M2 : DWORD ;
  COUNT_M3 : DWORD ;
  COUNT_M4 : DWORD ;
  COUNT_M5 : DWORD ;
  NR_MAX_M : DINT ;	//NR MAX FUNZIONI IN DINT
END_VAR
BEGIN
NETWORK
TITLE = DECODIFICA MAX 130 FUNZIONI OCCUPA M220.0 AD M235.7
      L     #NR_MAX_DECOD;
      ITD;
      T     #NR_MAX_M;
// _________________________ VERIFICA PRIMA M
      L     #VALORE_CODICE_M1;
      L     #NR_MAX_M;
      >D;
      O(;
      L     #VALORE_CODICE_M1;
      L     0;
      ==D;
      );
      JC    M001;
      L     P#220.0;
      T     #COUNT_M1;
      L     #COUNT_M1;
      L     #VALORE_CODICE_M1;
      +D;
      T     #COUNT_M1;
      =     M [#COUNT_M1];
M001: NOP   0;
//_________________________ VERIFICA SECONDA M
      L     #VALORE_CODICE_M2;
      L     #NR_MAX_M;
      >D;
      O(;
      L     #VALORE_CODICE_M2;
      L     0;
      ==D;
      );
      JC    M002;
      L     P#220.0;
      T     #COUNT_M2;
      L     #COUNT_M2;
      L     #VALORE_CODICE_M2;
      +D;
      T     #COUNT_M2;
      =     M [#COUNT_M2];
M002: NOP   0;
//_________________________ VERIFICA TERZA M
      L     #VALORE_CODICE_M3;
      L     #NR_MAX_M;
      >D;
      O(;
      L     #VALORE_CODICE_M3;
      L     0;
      ==D;
      );
      JC    M003;
      L     P#220.0;
      T     #COUNT_M3;
      L     #COUNT_M3;
      L     #VALORE_CODICE_M3;
      +D;
      T     #COUNT_M3;
      =     M [#COUNT_M3];
M003: NOP   0;
//_________________________ VERIFICA QUARTA M
      L     #VALORE_CODICE_M4;
      L     #NR_MAX_M;
      >D;
      O(;
      L     #VALORE_CODICE_M4;
      L     0;
      ==D;
      );
      JC    M004;
      L     P#220.0;
      T     #COUNT_M4;
      L     #COUNT_M4;
      L     #VALORE_CODICE_M4;
      +D;
      T     #COUNT_M4;
      =     M [#COUNT_M4];
M004: NOP   0;
//_________________________ VERIFICA QUINTA M
      L     #VALORE_CODICE_M5;
      L     #NR_MAX_M;
      >D;
      O(;
      L     #VALORE_CODICE_M5;
      L     0;
      ==D;
      );
      JC    M005;
      L     P#220.0;
      T     #COUNT_M5;
      L     #COUNT_M5;
      L     #VALORE_CODICE_M5;
      +D;
      T     #COUNT_M5;
      =     M [#COUNT_M5];
M005: NOP   0;
      L     0;
      T     "Chan1".M1;
      T     "Chan1".M2;
      T     "Chan1".M3;
      T     "Chan1".M4;
      T     "Chan1".M5;
//________________________ FUNZIONE M PRESENTE
      L     MW 218;
      L     0;
      <>I;
      O(;
      L     MD 220;
      L     0;
      <>D;
      );
      O(;
      L     MD 224;
      L     0;
      <>D;
      );
      O(;
      L     MD 228;
      L     0;
      <>D;
      );
      O(;
      L     MD 232;
      L     0;
      <>D;
      );
      =     #M_ATTIVA;
// ___________________________ TACITAZIONE DI RESET
      A     "Chan1".A_Reset;
      JCN   RESE;
      L     0;
      T     MW 218;
      T     MD 220;
      T     MD 224;
      T     MD 228;
      T     MD 232;
RESE: NOP   0;
END_FUNCTION

FUNCTION "FC Gestione Allarmi" : VOID	// FC 99
TITLE = Gestione Allarmi Macchina
AUTHOR : Asamec
VERSION : 0.1
VAR_OUTPUT
  BloccoLettura : BOOL ;	//da 510216 a 510315 (DB2.DBX8.0 - DB2.DBX 11.7)
  BloccoAssi : BOOL ;	//da 511100 a 511215 (DB2.DBX12.0 - DB2.DBX15.7)
  BloccoMandrino : BOOL ;	//da 600100 a 600115 (DB2.DBX 144.0 - DB2.DBX 145.7)
  BloccoAssiMandrino : BOOL ;	//da 510000 a 510215 (DB2.DBX0.0 - DB2.DBX7.7
  BloccoRipartenza : BOOL ;	//da 700100 a 700131 (DB2.DBX188.0 - DB2.DBX191.7)
  Messaggio : BOOL ;	//da 700000 a 700063  (DB2.DBX180.0 - DB2.DBX187.7)
END_VAR
BEGIN
NETWORK
TITLE = Blocco Lettura
      L     DB2.DBD 8;
      L     0;
      <>D;
      =     #BloccoLettura;
NETWORK
TITLE = Blocco Assi
      L     DB2.DBD 12;
      L     0;
      <>D;
      =     #BloccoAssi;
NETWORK
TITLE = Blocco Mandrino
      L     "DB Allarmi".Asse1_Feed_Stop;
      L     0;
      <>I;
      =     #BloccoMandrino;
NETWORK
TITLE = Blocco Assi e Mandrino
      L     DB2.DBD 0;
      L     0;
      <>D;
      O(;
      L     DB2.DBD 4;
      L     0;
      <>D;
      );
      =     #BloccoAssiMandrino;
NETWORK
TITLE = BloccoRipartenza
      L     DB2.DBD 188;
      L     0;
      <>D;
      =     #BloccoRipartenza;
NETWORK
TITLE = Messaggio
      L     DB2.DBD 180;
      L     0;
      <>D;
      O;
      L     DB2.DBD 184;
      L     0;
      <>D;
      =     #Messaggio;
END_FUNCTION

FUNCTION "FC Generali" : VOID	// FC 100
AUTHOR : Asamec
VERSION : 0.1
BEGIN
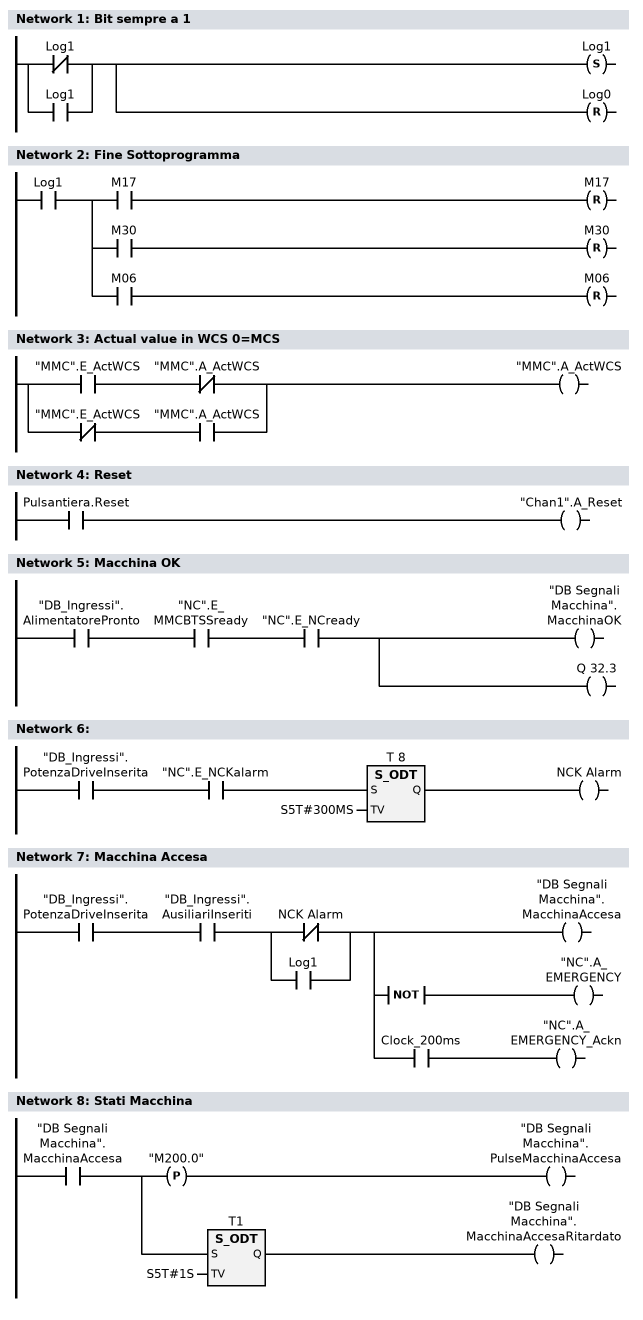
NETWORK
TITLE = Bit sempre a 1
      ON    "Log1";
      O     "Log1";
      S     "Log1";
      R     "Log0";
NETWORK
TITLE = Fine Sottoprogramma
      A     "Log1";
      =     L 0.0;
      A     L 0.0;
      A     "M17";
      R     "M17";
      A     L 0.0;
      A     "M30";
      R     "M30";
      A     L 0.0;
      A     "M06";
      R     "M06";
NETWORK
TITLE = Actual value in WCS 0=MCS
      A     "MMC".E_ActWCS;
      AN    "MMC".A_ActWCS;
      O;
      AN    "MMC".E_ActWCS;
      A     "MMC".A_ActWCS;
      =     "MMC".A_ActWCS;
NETWORK
TITLE = Reset
      A     "Pulsantiera.Reset";
      =     "Chan1".A_Reset;
NETWORK
TITLE = Macchina OK
      A     "DB_Ingressi".AlimentatorePronto;
      A     "NC".E_MMCBTSSready;
      A     "NC".E_NCready;
      =     "DB Segnali Macchina".MacchinaOK;
      =     Q 32.3;
NETWORK
TITLE =
      A     "DB_Ingressi".PotenzaDriveInserita;
      A     "NC".E_NCKalarm;
      L     S5T#300MS;
      SD    T 8;
      NOP   0;
      NOP   0;
      NOP   0;
      A     T 8;
      =     "NCK Alarm";
NETWORK
TITLE = Macchina Accesa
      A     "DB_Ingressi".PotenzaDriveInserita;
      A     "DB_Ingressi".AusiliariInseriti;
      A(;
      ON    "NCK Alarm";
      O     "Log1";
      );
      =     L 0.0;
      A     L 0.0;
      BLD   102;
      =     "DB Segnali Macchina".MacchinaAccesa;
      A     L 0.0;
      NOT;
      =     "NC".A_EMERGENCY;
      A     L 0.0;
      A     "Clock_200ms";
      =     "NC".A_EMERGENCY_Ackn;
NETWORK
TITLE = Stati Macchina
      A     "DB Segnali Macchina".MacchinaAccesa;
      =     L 0.0;
      A     L 0.0;
      FP    "M200.0";
      =     "DB Segnali Macchina".PulseMacchinaAccesa;
      A     L 0.0;
      L     S5T#1S;
      SD    "T1";
      NOP   0;
      NOP   0;
      NOP   0;
      A     "T1";
      =     "DB Segnali Macchina".MacchinaAccesaRitardato;
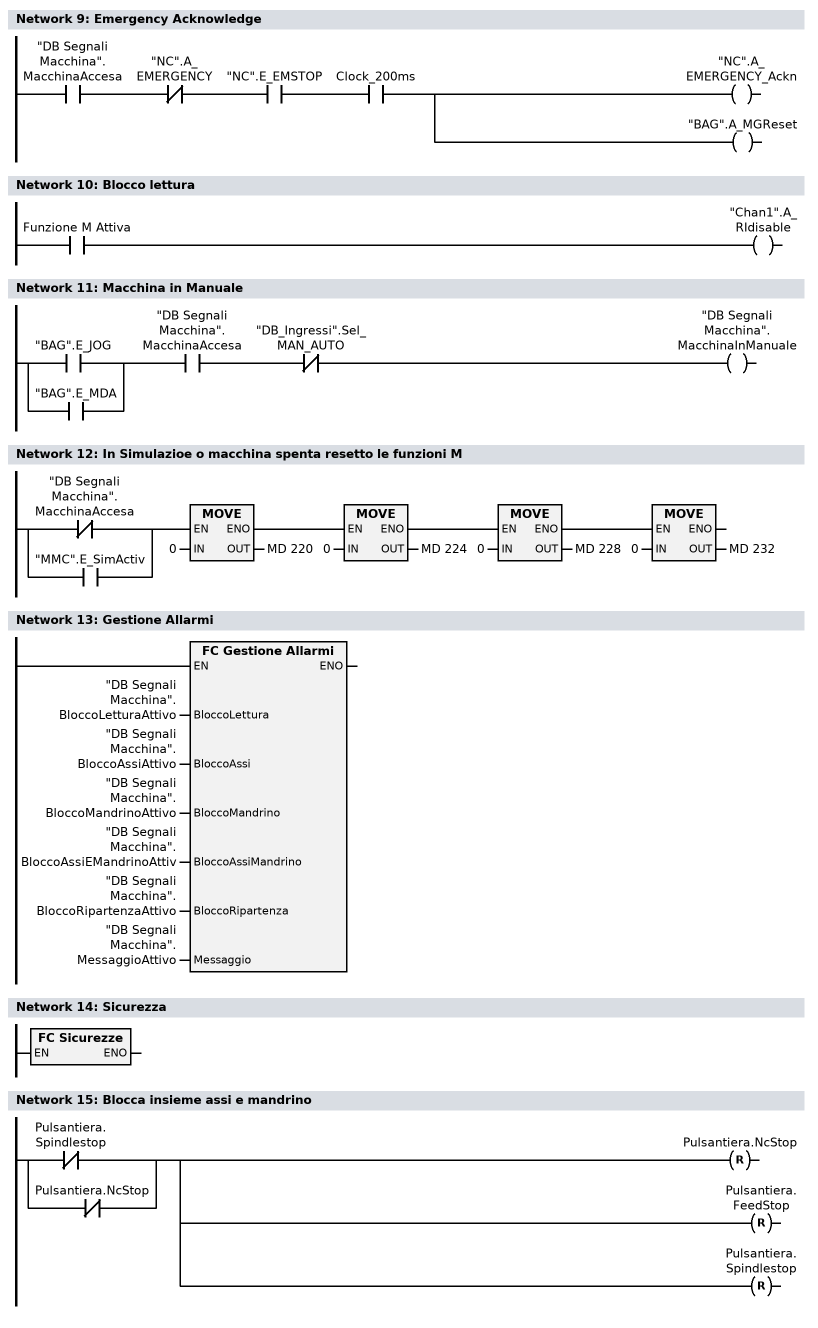
NETWORK
TITLE = Emergency Acknowledge
      A     "DB Segnali Macchina".MacchinaAccesa;
      AN    "NC".A_EMERGENCY;
      A     "NC".E_EMSTOP;
      A     "Clock_200ms";
      =     "NC".A_EMERGENCY_Ackn;
      =     "BAG".A_MGReset;
NETWORK
TITLE = Blocco lettura
      A     "Funzione M Attiva";
      =     "Chan1".A_RIdisable;
NETWORK
TITLE = Macchina in Manuale
      A(;
      O     "BAG".E_JOG;
      O     "BAG".E_MDA;
      );
      A     "DB Segnali Macchina".MacchinaAccesa;
      AN    "DB_Ingressi".Sel_MAN_AUTO;
      =     "DB Segnali Macchina".MacchinaInManuale;
NETWORK
TITLE = In Simulazioe o macchina spenta resetto le funzioni M
      A(;
      A(;
      A(;
      A(;
      ON    "DB Segnali Macchina".MacchinaAccesa;
      O     "MMC".E_SimActiv;
      );
      JNB   _001;
      L     0;
      T     MD 220;
      SET;
      SAVE;
      CLR;
_001: A     BR;
      );
      JNB   _002;
      L     0;
      T     MD 224;
      SET;
      SAVE;
      CLR;
_002: A     BR;
      );
      JNB   _003;
      L     0;
      T     MD 228;
      SET;
      SAVE;
      CLR;
_003: A     BR;
      );
      JNB   _004;
      L     0;
      T     MD 232;
_004: NOP   0;
NETWORK
TITLE = Gestione Allarmi
      CALL  "FC Gestione Allarmi" (
           BloccoLettura            := "DB Segnali Macchina".BloccoLetturaAttivo,
           BloccoAssi               := "DB Segnali Macchina".BloccoAssiAttivo,
           BloccoMandrino           := "DB Segnali Macchina".BloccoMandrinoAttivo,
           BloccoAssiMandrino       := "DB Segnali Macchina".BloccoAssiEMandrinoAttiv,
           BloccoRipartenza         := "DB Segnali Macchina".BloccoRipartenzaAttivo,
           Messaggio                := "DB Segnali Macchina".MessaggioAttivo);
      NOP   0;
NETWORK
TITLE = Sicurezza
      CALL  "FC Sicurezze";
      NOP   0;
NETWORK
TITLE = Blocca insieme assi e mandrino
      ON    "Pulsantiera.Spindlestop";
      ON    "Pulsantiera.NcStop";
      R     "Pulsantiera.NcStop";
      R     "Pulsantiera.FeedStop";
      R     "Pulsantiera.Spindlestop";
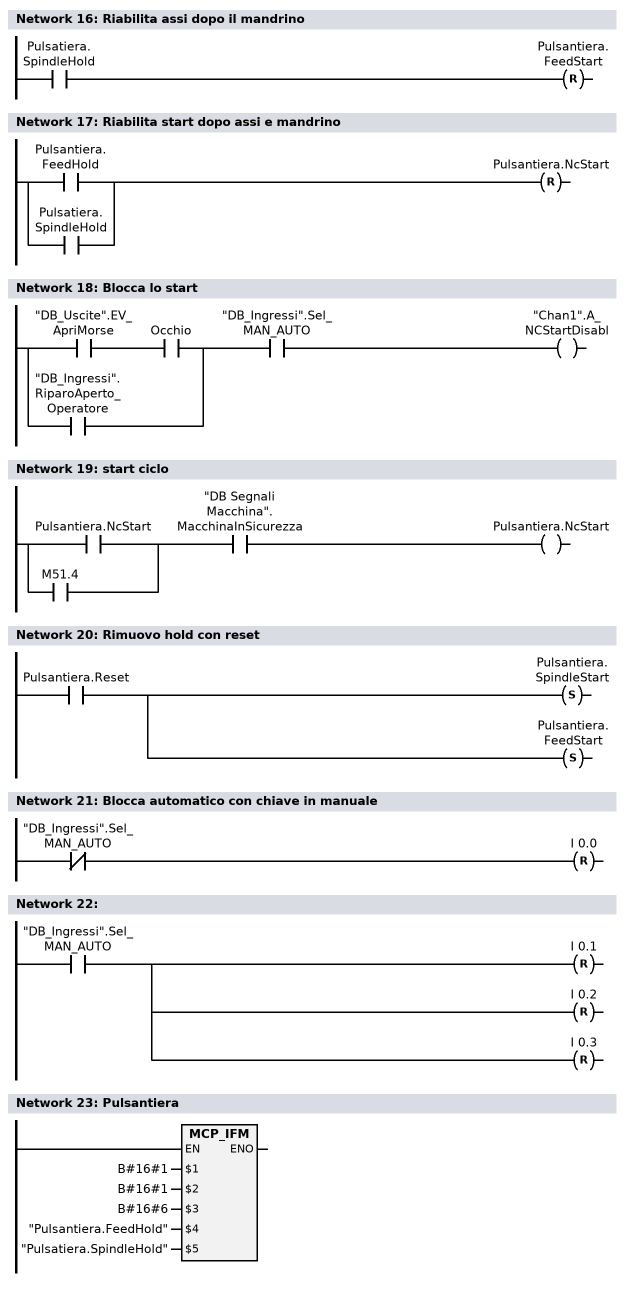
NETWORK
TITLE = Riabilita assi dopo il mandrino
      A     "Pulsatiera.SpindleHold";
      R     "Pulsantiera.FeedStart";
NETWORK
TITLE = Riabilita start dopo assi e mandrino
      O     "Pulsantiera.FeedHold";
      O     "Pulsatiera.SpindleHold";
      R     "Pulsantiera.NcStart";
NETWORK
TITLE = Blocca lo start
      A(;
      A     "DB_Uscite".EV_ApriMorse;
      A     "Occhio";
      O     "DB_Ingressi".RiparoAperto_Operatore;
      );
      A     "DB_Ingressi".Sel_MAN_AUTO;
      =     "Chan1".A_NCStartDisabl;
NETWORK
TITLE = start ciclo
      A(;
      O     "Pulsantiera.NcStart";
      O     "M51.4";
      );
      A     "DB Segnali Macchina".MacchinaInSicurezza;
      =     "Pulsantiera.NcStart";
NETWORK
TITLE = Rimuovo hold con reset
      A     "Pulsantiera.Reset";
      S     "Pulsantiera.SpindleStart";
      S     "Pulsantiera.FeedStart";
NETWORK
TITLE = Blocca automatico con chiave in manuale
      AN    "DB_Ingressi".Sel_MAN_AUTO;
      R     I 0.0;
NETWORK
TITLE =
      A     "DB_Ingressi".Sel_MAN_AUTO;
      R     I 0.1;
      R     I 0.2;
      R     I 0.3;
NETWORK
TITLE = Pulsantiera
      CALL  "MCP_IFM" (
           $1                       := B#16#1,
           $2                       := B#16#1,
           $3                       := B#16#6,
           $4                       := "Pulsantiera.FeedHold",
           $5                       := "Pulsatiera.SpindleHold");
      NOP   0;
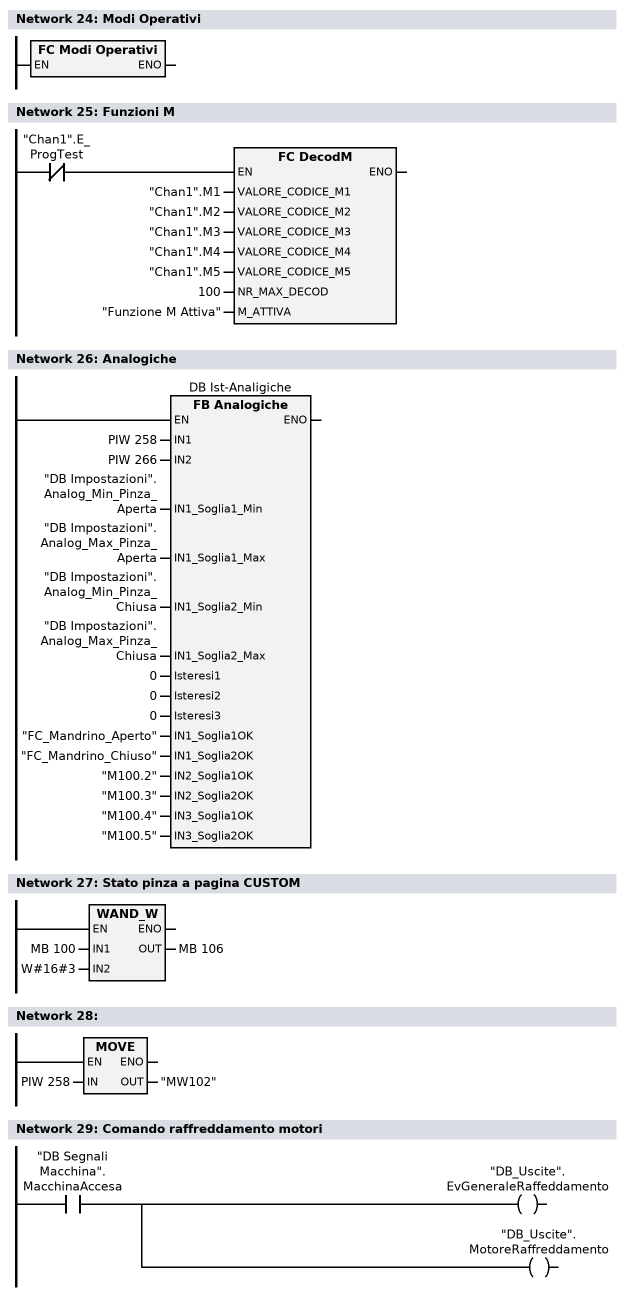
NETWORK
TITLE = Modi Operativi
      CALL  "FC Modi Operativi";
      NOP   0;
NETWORK
TITLE = Funzioni M
      AN    "Chan1".E_ProgTest;
      JNB   _005;
      CALL  "FC DecodM" (
           VALORE_CODICE_M1         := "Chan1".M1,
           VALORE_CODICE_M2         := "Chan1".M2,
           VALORE_CODICE_M3         := "Chan1".M3,
           VALORE_CODICE_M4         := "Chan1".M4,
           VALORE_CODICE_M5         := "Chan1".M5,
           NR_MAX_DECOD             := 100,
           M_ATTIVA                 := "Funzione M Attiva");
_005: NOP   0;
NETWORK
TITLE = Analogiche
      CALL  "FB Analogiche" , "DB Ist-Analigiche" (
           IN1                      := PIW 258,
           IN2                      := PIW 266,
           IN1_Soglia1_Min          := "DB Impostazioni".Analog_Min_Pinza_Aperta,
           IN1_Soglia1_Max          := "DB Impostazioni".Analog_Max_Pinza_Aperta,
           IN1_Soglia2_Min          := "DB Impostazioni".Analog_Min_Pinza_Chiusa,
           IN1_Soglia2_Max          := "DB Impostazioni".Analog_Max_Pinza_Chiusa,
           Isteresi1                := 0,
           Isteresi2                := 0,
           Isteresi3                := 0,
           IN1_Soglia1OK            := "FC_Mandrino_Aperto",
           IN1_Soglia2OK            := "FC_Mandrino_Chiuso",
           IN2_Soglia1OK            := "M100.2",
           IN2_Soglia2OK            := "M100.3",
           IN3_Soglia1OK            := "M100.4",
           IN3_Soglia2OK            := "M100.5");
      NOP   0;
NETWORK
TITLE = Stato pinza a pagina CUSTOM
      L     MB 100;
      L     W#16#3;
      AW;
      T     MB 106;
NETWORK
TITLE =
      L     PIW 258;
      T     "MW102";
      NOP   0;
NETWORK
TITLE = Comando raffreddamento motori
      A     "DB Segnali Macchina".MacchinaAccesa;
      =     "DB_Uscite".EvGeneraleRaffeddamento;
      =     "DB_Uscite".MotoreRaffreddamento;
END_FUNCTION

FUNCTION "FC Ingressi" : VOID	// FC 101
AUTHOR : Asamec
VERSION : 0.1
BEGIN
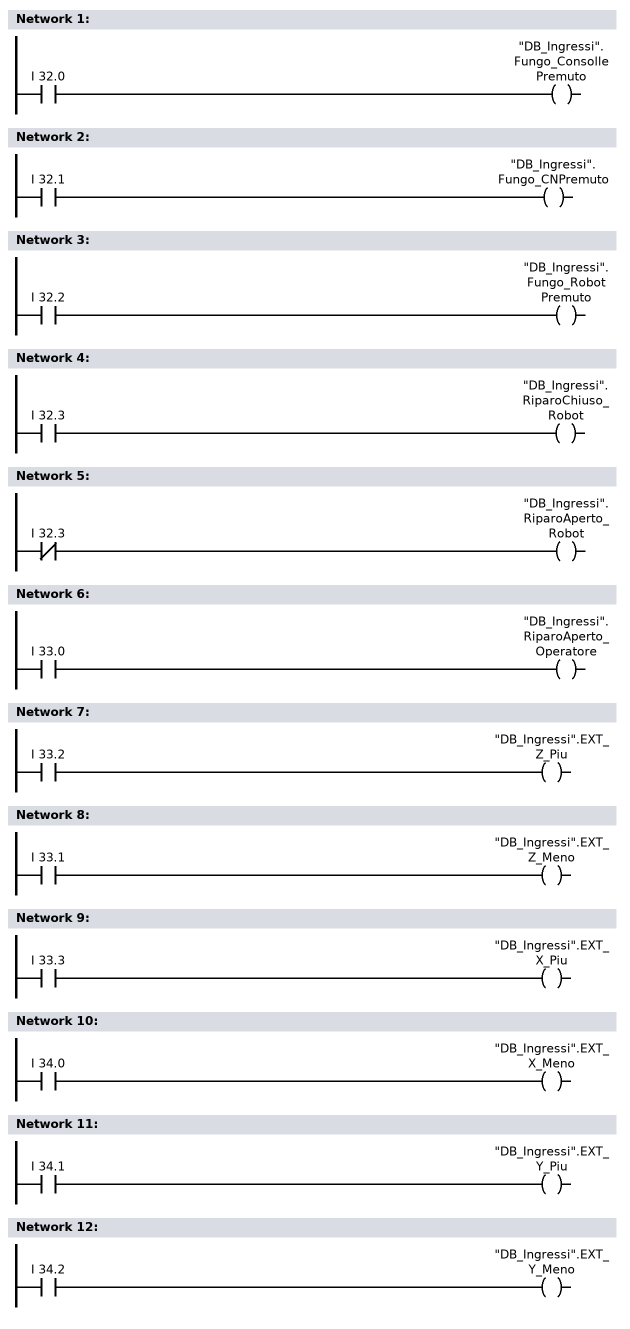
NETWORK
TITLE =
      A     I 32.0;
      =     "DB_Ingressi".Fungo_ConsollePremuto;
NETWORK
TITLE =
      A     I 32.1;
      =     "DB_Ingressi".Fungo_CNPremuto;
NETWORK
TITLE =
      A     I 32.2;
      =     "DB_Ingressi".Fungo_RobotPremuto;
NETWORK
TITLE =
      A     I 32.3;
      =     "DB_Ingressi".RiparoChiuso_Robot;
NETWORK
TITLE =
      AN    I 32.3;
      =     "DB_Ingressi".RiparoAperto_Robot;
NETWORK
TITLE =
      A     I 33.0;
      =     "DB_Ingressi".RiparoAperto_Operatore;
NETWORK
TITLE =
      A     I 33.2;
      =     "DB_Ingressi".EXT_Z_Piu;
NETWORK
TITLE =
      A     I 33.1;
      =     "DB_Ingressi".EXT_Z_Meno;
NETWORK
TITLE =
      A     I 33.3;
      =     "DB_Ingressi".EXT_X_Piu;
NETWORK
TITLE =
      A     I 34.0;
      =     "DB_Ingressi".EXT_X_Meno;
NETWORK
TITLE =
      A     I 34.1;
      =     "DB_Ingressi".EXT_Y_Piu;
NETWORK
TITLE =
      A     I 34.2;
      =     "DB_Ingressi".EXT_Y_Meno;
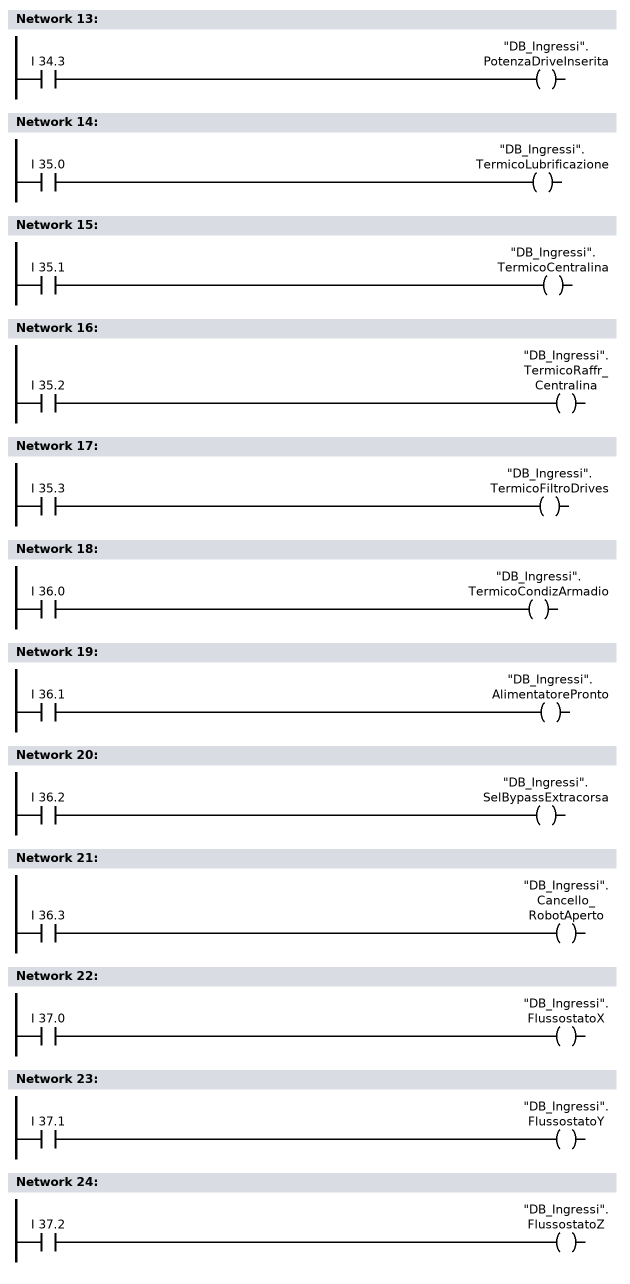
NETWORK
TITLE =
      A     I 34.3;
      =     "DB_Ingressi".PotenzaDriveInserita;
NETWORK
TITLE =
      A     I 35.0;
      =     "DB_Ingressi".TermicoLubrificazione;
NETWORK
TITLE =
      A     I 35.1;
      =     "DB_Ingressi".TermicoCentralina;
NETWORK
TITLE =
      A     I 35.2;
      =     "DB_Ingressi".TermicoRaffr_Centralina;
NETWORK
TITLE =
      A     I 35.3;
      =     "DB_Ingressi".TermicoFiltroDrives;
NETWORK
TITLE =
      A     I 36.0;
      =     "DB_Ingressi".TermicoCondizArmadio;
NETWORK
TITLE =
      A     I 36.1;
      =     "DB_Ingressi".AlimentatorePronto;
NETWORK
TITLE =
      A     I 36.2;
      =     "DB_Ingressi".SelBypassExtracorsa;
NETWORK
TITLE =
      A     I 36.3;
      =     "DB_Ingressi".Cancello_RobotAperto;
NETWORK
TITLE =
      A     I 37.0;
      =     "DB_Ingressi".FlussostatoX;
NETWORK
TITLE =
      A     I 37.1;
      =     "DB_Ingressi".FlussostatoY;
NETWORK
TITLE =
      A     I 37.2;
      =     "DB_Ingressi".FlussostatoZ;
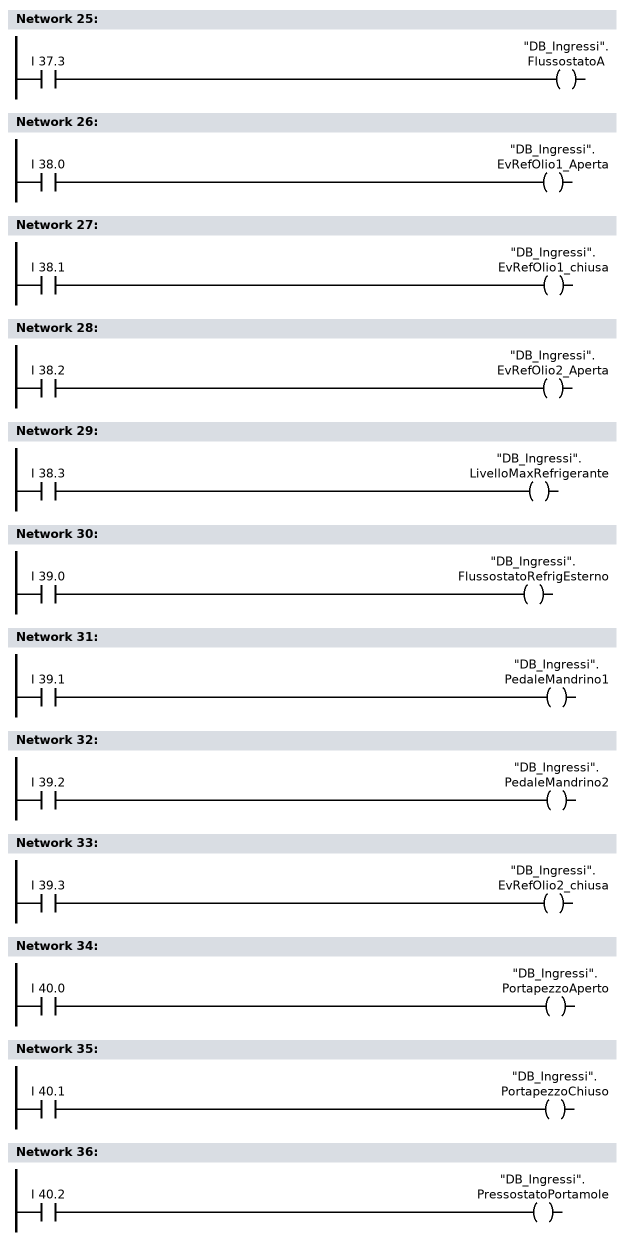
NETWORK
TITLE =
      A     I 37.3;
      =     "DB_Ingressi".FlussostatoA;
NETWORK
TITLE =
      A     I 38.0;
      =     "DB_Ingressi".EvRefOlio1_Aperta;
NETWORK
TITLE =
      A     I 38.1;
      =     "DB_Ingressi".EvRefOlio1_chiusa;
NETWORK
TITLE =
      A     I 38.2;
      =     "DB_Ingressi".EvRefOlio2_Aperta;
NETWORK
TITLE =
      A     I 38.3;
      =     "DB_Ingressi".LivelloMaxRefrigerante;
NETWORK
TITLE =
      A     I 39.0;
      =     "DB_Ingressi".FlussostatoRefrigEsterno;
NETWORK
TITLE =
      A     I 39.1;
      =     "DB_Ingressi".PedaleMandrino1;
NETWORK
TITLE =
      A     I 39.2;
      =     "DB_Ingressi".PedaleMandrino2;
NETWORK
TITLE =
      A     I 39.3;
      =     "DB_Ingressi".EvRefOlio2_chiusa;
NETWORK
TITLE =
      A     I 40.0;
      =     "DB_Ingressi".PortapezzoAperto;
NETWORK
TITLE =
      A     I 40.1;
      =     "DB_Ingressi".PortapezzoChiuso;
NETWORK
TITLE =
      A     I 40.2;
      =     "DB_Ingressi".PressostatoPortamole;
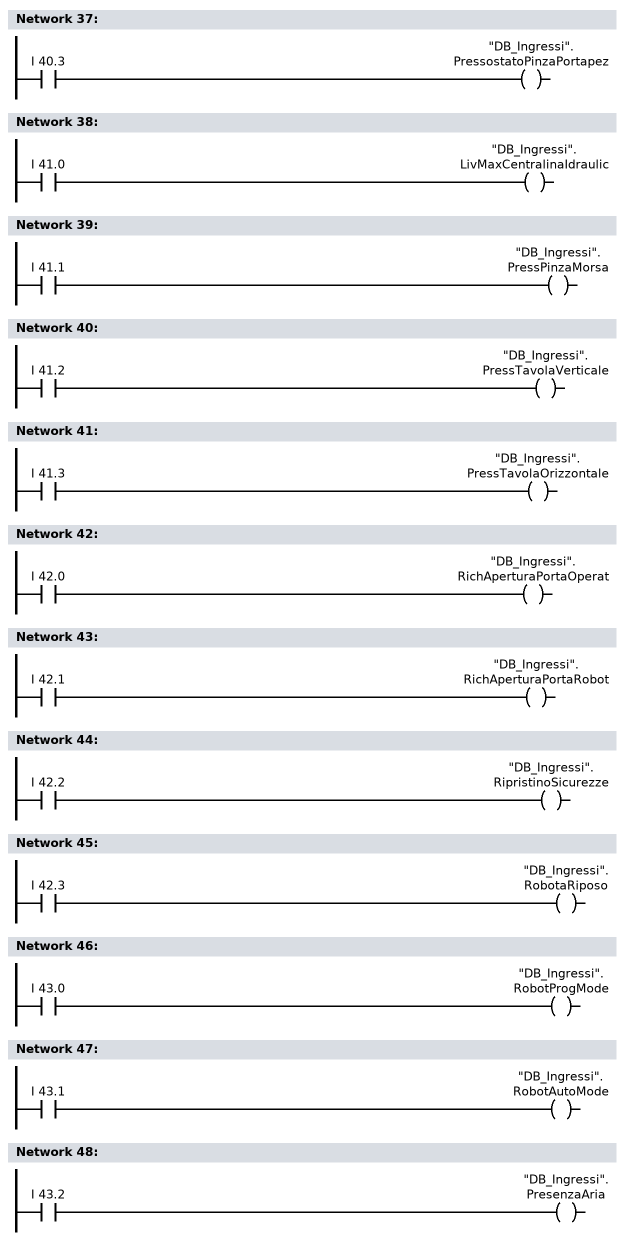
NETWORK
TITLE =
      A     I 40.3;
      =     "DB_Ingressi".PressostatoPinzaPortapez;
NETWORK
TITLE =
      A     I 41.0;
      =     "DB_Ingressi".LivMaxCentralinaIdraulic;
NETWORK
TITLE =
      A     I 41.1;
      =     "DB_Ingressi".PressPinzaMorsa;
NETWORK
TITLE =
      A     I 41.2;
      =     "DB_Ingressi".PressTavolaVerticale;
NETWORK
TITLE =
      A     I 41.3;
      =     "DB_Ingressi".PressTavolaOrizzontale;
NETWORK
TITLE =
      A     I 42.0;
      =     "DB_Ingressi".RichAperturaPortaOperat;
NETWORK
TITLE =
      A     I 42.1;
      =     "DB_Ingressi".RichAperturaPortaRobot;
NETWORK
TITLE =
      A     I 42.2;
      =     "DB_Ingressi".RipristinoSicurezze;
NETWORK
TITLE =
      A     I 42.3;
      =     "DB_Ingressi".RobotaRiposo;
NETWORK
TITLE =
      A     I 43.0;
      =     "DB_Ingressi".RobotProgMode;
NETWORK
TITLE =
      A     I 43.1;
      =     "DB_Ingressi".RobotAutoMode;
NETWORK
TITLE =
      A     I 43.2;
      =     "DB_Ingressi".PresenzaAria;
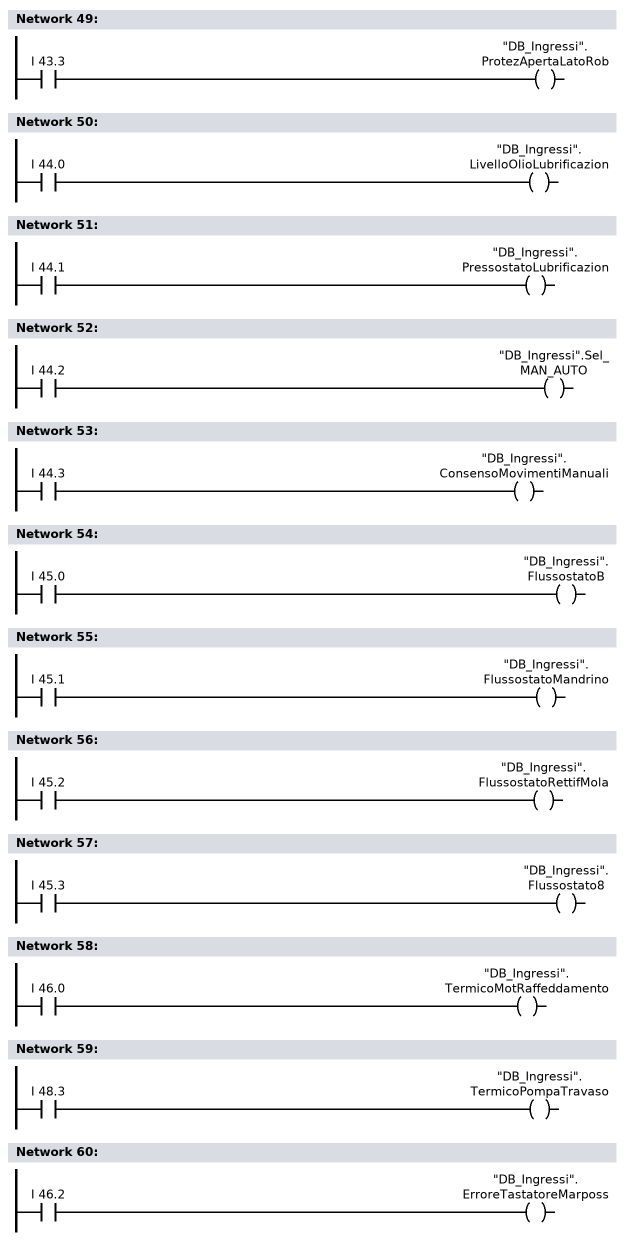
NETWORK
TITLE =
      A     I 43.3;
      =     "DB_Ingressi".ProtezApertaLatoRob;
NETWORK
TITLE =
      A     I 44.0;
      =     "DB_Ingressi".LivelloOlioLubrificazion;
NETWORK
TITLE =
      A     I 44.1;
      =     "DB_Ingressi".PressostatoLubrificazion;
NETWORK
TITLE =
      A     I 44.2;
      =     "DB_Ingressi".Sel_MAN_AUTO;
NETWORK
TITLE =
      A     I 44.3;
      =     "DB_Ingressi".ConsensoMovimentiManuali;
NETWORK
TITLE =
      A     I 45.0;
      =     "DB_Ingressi".FlussostatoB;
NETWORK
TITLE =
      A     I 45.1;
      =     "DB_Ingressi".FlussostatoMandrino;
NETWORK
TITLE =
      A     I 45.2;
      =     "DB_Ingressi".FlussostatoRettifMola;
NETWORK
TITLE =
      A     I 45.3;
      =     "DB_Ingressi".Flussostato8;
NETWORK
TITLE =
      A     I 46.0;
      =     "DB_Ingressi".TermicoMotRaffeddamento;
NETWORK
TITLE =
      A     I 48.3;
      =     "DB_Ingressi".TermicoPompaTravaso;
NETWORK
TITLE =
      A     I 46.2;
      =     "DB_Ingressi".ErroreTastatoreMarposs;
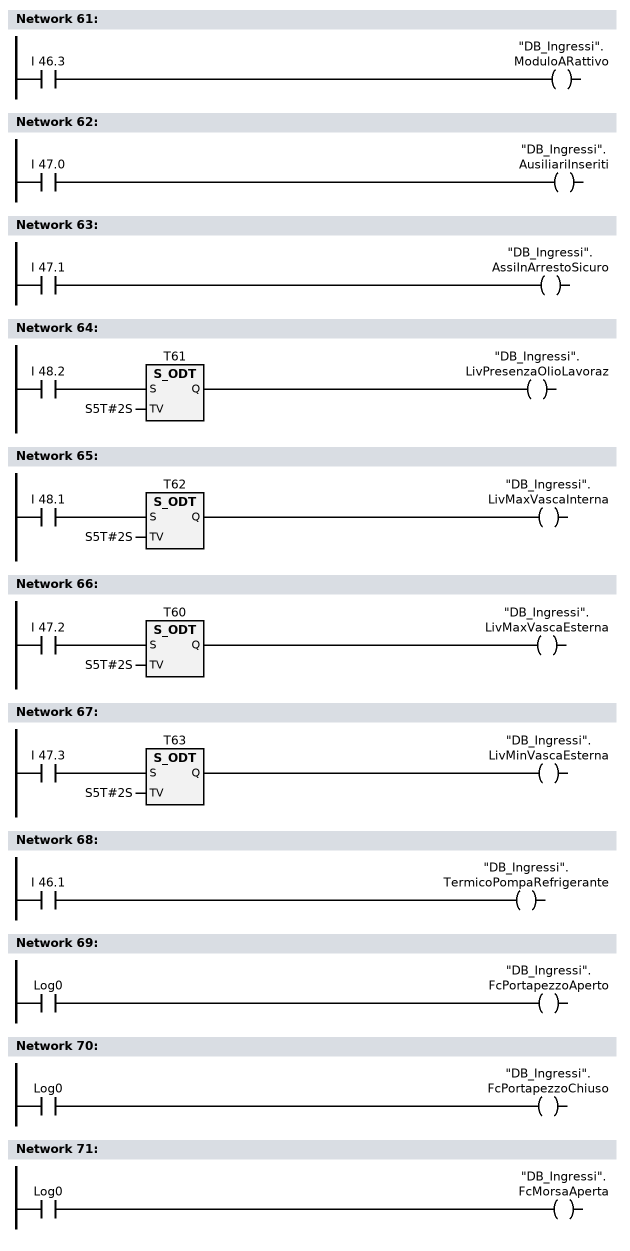
NETWORK
TITLE =
      A     I 46.3;
      =     "DB_Ingressi".ModuloARattivo;
NETWORK
TITLE =
      A     I 47.0;
      =     "DB_Ingressi".AusiliariInseriti;
NETWORK
TITLE =
      A     I 47.1;
      =     "DB_Ingressi".AssiInArrestoSicuro;
NETWORK
TITLE =
      A     I 48.2;
      L     S5T#2S;
      SD    "T61";
      NOP   0;
      NOP   0;
      NOP   0;
      A     "T61";
      =     "DB_Ingressi".LivPresenzaOlioLavoraz;
NETWORK
TITLE =
      A     I 48.1;
      L     S5T#2S;
      SD    "T62";
      NOP   0;
      NOP   0;
      NOP   0;
      A     "T62";
      =     "DB_Ingressi".LivMaxVascaInterna;
NETWORK
TITLE =
      A     I 47.2;
      L     S5T#2S;
      SD    "T60";
      NOP   0;
      NOP   0;
      NOP   0;
      A     "T60";
      =     "DB_Ingressi".LivMaxVascaEsterna;
NETWORK
TITLE =
      A     I 47.3;
      L     S5T#2S;
      SD    "T63";
      NOP   0;
      NOP   0;
      NOP   0;
      A     "T63";
      =     "DB_Ingressi".LivMinVascaEsterna;
NETWORK
TITLE =
      A     I 46.1;
      =     "DB_Ingressi".TermicoPompaRefrigerante;
NETWORK
TITLE =
      A     "Log0";
      =     "DB_Ingressi".FcPortapezzoAperto;
NETWORK
TITLE =
      A     "Log0";
      =     "DB_Ingressi".FcPortapezzoChiuso;
NETWORK
TITLE =
      A     "Log0";
      =     "DB_Ingressi".FcMorsaAperta;
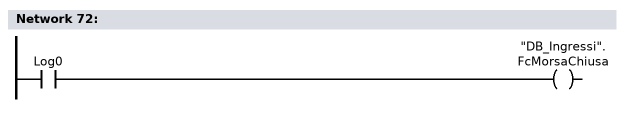
NETWORK
TITLE =
      A     "Log0";
      =     "DB_Ingressi".FcMorsaChiusa;
END_FUNCTION

FUNCTION "FC Uscite" : VOID	// FC 102
AUTHOR : Asamec
VERSION : 0.1
BEGIN
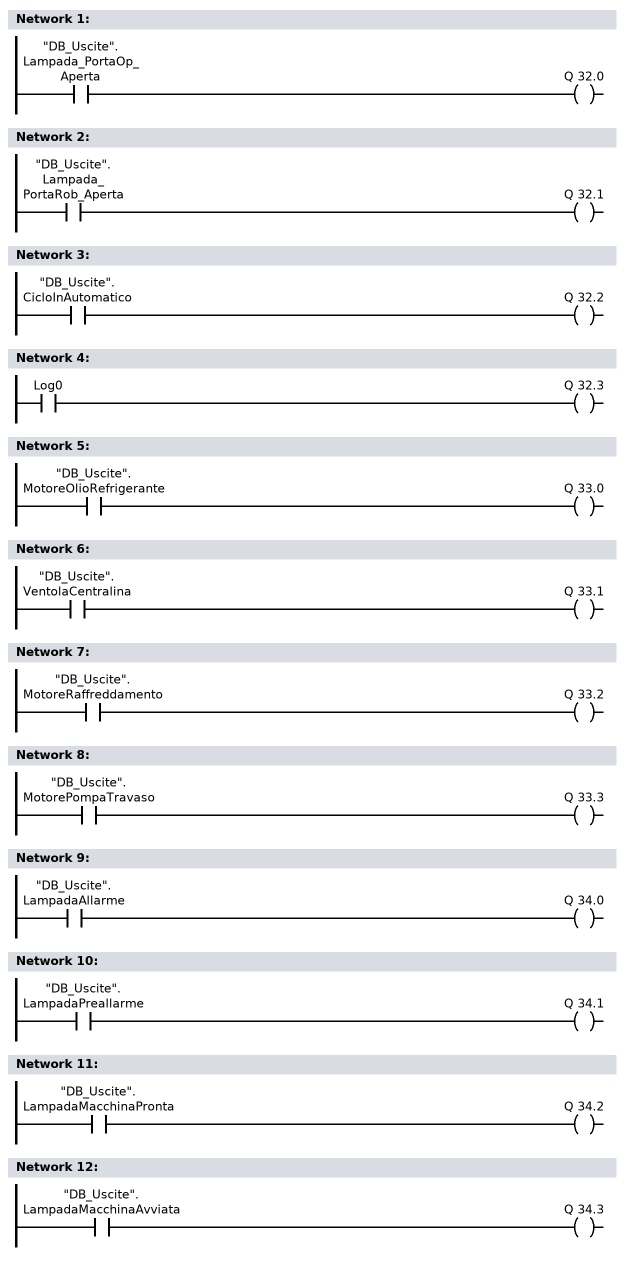
NETWORK
TITLE =
      A     "DB_Uscite".Lampada_PortaOp_Aperta;
      =     Q 32.0;
NETWORK
TITLE =
      A     "DB_Uscite".Lampada_PortaRob_Aperta;
      =     Q 32.1;
NETWORK
TITLE =
      A     "DB_Uscite".CicloInAutomatico;
      =     Q 32.2;
NETWORK
TITLE =
      A     "Log0";
      =     Q 32.3;
NETWORK
TITLE =
      A     "DB_Uscite".MotoreOlioRefrigerante;
      =     Q 33.0;
NETWORK
TITLE =
      A     "DB_Uscite".VentolaCentralina;
      =     Q 33.1;
NETWORK
TITLE =
      A     "DB_Uscite".MotoreRaffreddamento;
      =     Q 33.2;
NETWORK
TITLE =
      A     "DB_Uscite".MotorePompaTravaso;
      =     Q 33.3;
NETWORK
TITLE =
      A     "DB_Uscite".LampadaAllarme;
      =     Q 34.0;
NETWORK
TITLE =
      A     "DB_Uscite".LampadaPreallarme;
      =     Q 34.1;
NETWORK
TITLE =
      A     "DB_Uscite".LampadaMacchinaPronta;
      =     Q 34.2;
NETWORK
TITLE =
      A     "DB_Uscite".LampadaMacchinaAvviata;
      =     Q 34.3;
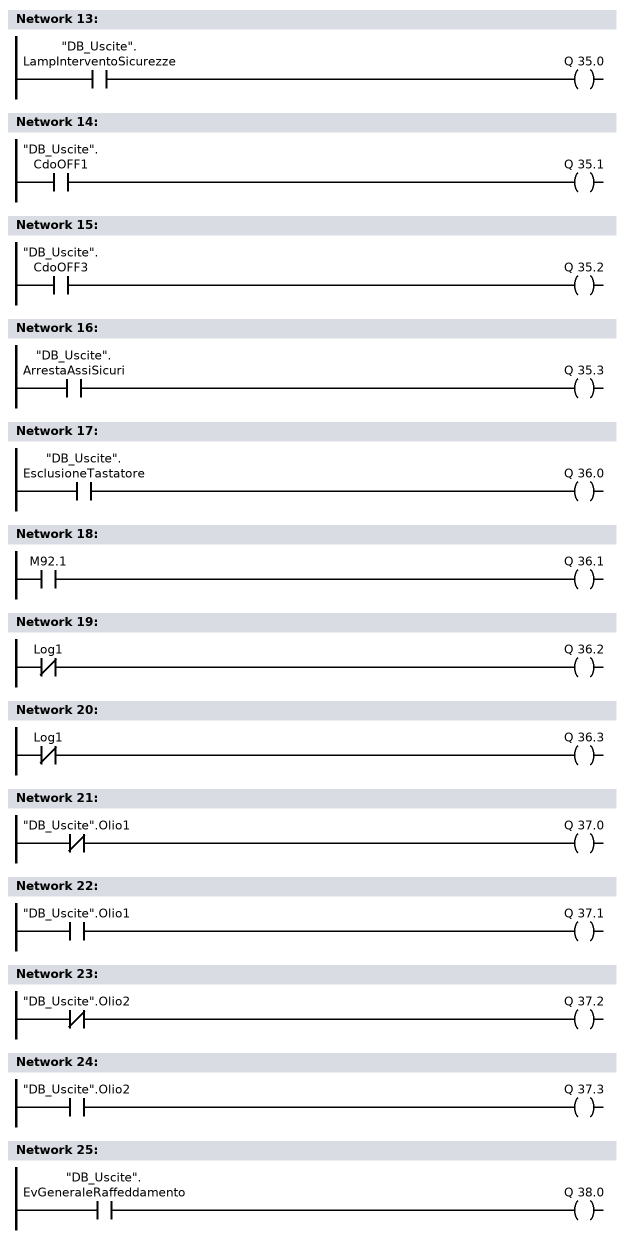
NETWORK
TITLE =
      A     "DB_Uscite".LampInterventoSicurezze;
      =     Q 35.0;
NETWORK
TITLE =
      A     "DB_Uscite".CdoOFF1;
      =     Q 35.1;
NETWORK
TITLE =
      A     "DB_Uscite".CdoOFF3;
      =     Q 35.2;
NETWORK
TITLE =
      A     "DB_Uscite".ArrestaAssiSicuri;
      =     Q 35.3;
NETWORK
TITLE =
      A     "DB_Uscite".EsclusioneTastatore;
      =     Q 36.0;
NETWORK
TITLE =
      A     "M92.1";
      =     Q 36.1;
NETWORK
TITLE =
      AN    "Log1";
      =     Q 36.2;
NETWORK
TITLE =
      AN    "Log1";
      =     Q 36.3;
NETWORK
TITLE =
      AN    "DB_Uscite".Olio1;
      =     Q 37.0;
NETWORK
TITLE =
      A     "DB_Uscite".Olio1;
      =     Q 37.1;
NETWORK
TITLE =
      AN    "DB_Uscite".Olio2;
      =     Q 37.2;
NETWORK
TITLE =
      A     "DB_Uscite".Olio2;
      =     Q 37.3;
NETWORK
TITLE =
      A     "DB_Uscite".EvGeneraleRaffeddamento;
      =     Q 38.0;
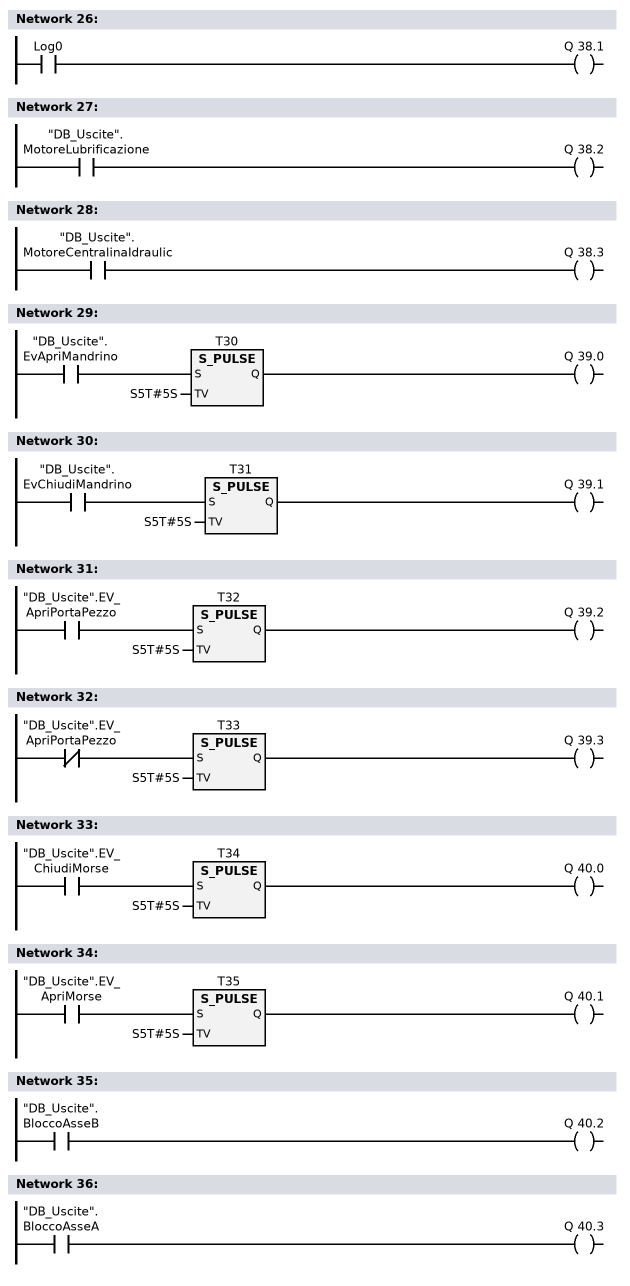
NETWORK
TITLE =
      A     "Log0";
      =     Q 38.1;
NETWORK
TITLE =
      A     "DB_Uscite".MotoreLubrificazione;
      =     Q 38.2;
NETWORK
TITLE =
      A     "DB_Uscite".MotoreCentralinaIdraulic;
      =     Q 38.3;
NETWORK
TITLE =
      A     "DB_Uscite".EvApriMandrino;
      L     S5T#5S;
      SP    "T30";
      NOP   0;
      NOP   0;
      NOP   0;
      A     "T30";
      =     Q 39.0;
NETWORK
TITLE =
      A     "DB_Uscite".EvChiudiMandrino;
      L     S5T#5S;
      SP    "T31";
      NOP   0;
      NOP   0;
      NOP   0;
      A     "T31";
      =     Q 39.1;
NETWORK
TITLE =
      A     "DB_Uscite".EV_ApriPortaPezzo;
      L     S5T#5S;
      SP    "T32";
      NOP   0;
      NOP   0;
      NOP   0;
      A     "T32";
      =     Q 39.2;
NETWORK
TITLE =
      AN    "DB_Uscite".EV_ApriPortaPezzo;
      L     S5T#5S;
      SP    "T33";
      NOP   0;
      NOP   0;
      NOP   0;
      A     "T33";
      =     Q 39.3;
NETWORK
TITLE =
      A     "DB_Uscite".EV_ChiudiMorse;
      L     S5T#5S;
      SP    "T34";
      NOP   0;
      NOP   0;
      NOP   0;
      A     "T34";
      =     Q 40.0;
NETWORK
TITLE =
      A     "DB_Uscite".EV_ApriMorse;
      L     S5T#5S;
      SP    "T35";
      NOP   0;
      NOP   0;
      NOP   0;
      A     "T35";
      =     Q 40.1;
NETWORK
TITLE =
      A     "DB_Uscite".BloccoAsseB;
      =     Q 40.2;
NETWORK
TITLE =
      A     "DB_Uscite".BloccoAsseA;
      =     Q 40.3;
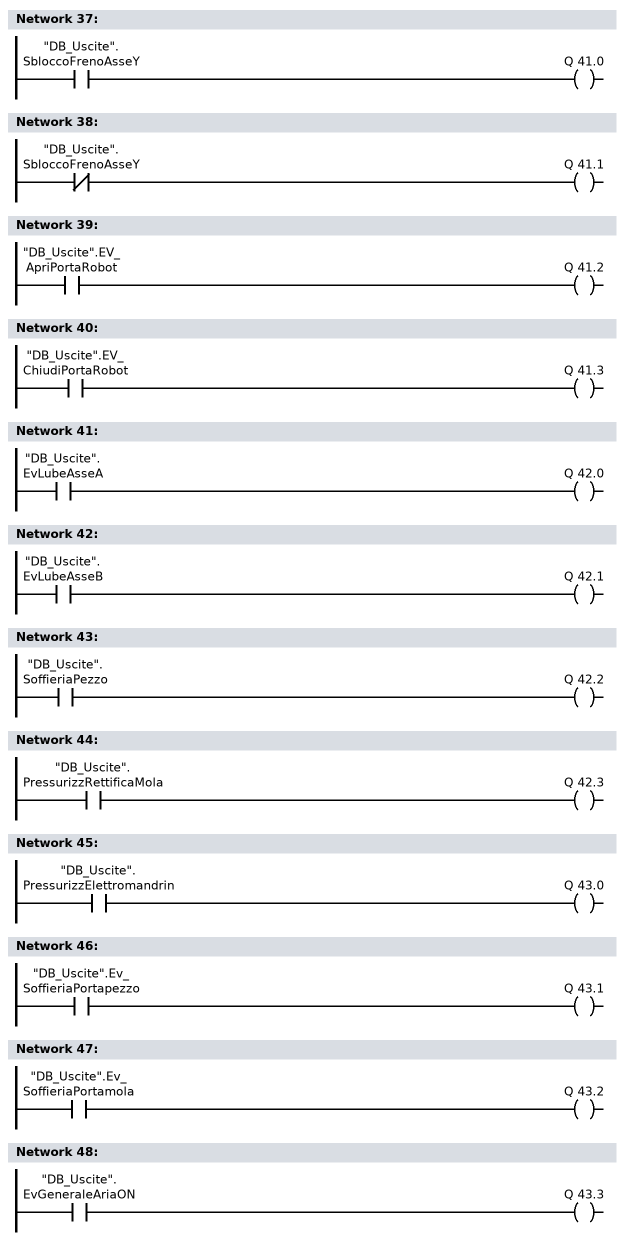
NETWORK
TITLE =
      A     "DB_Uscite".SbloccoFrenoAsseY;
      =     Q 41.0;
NETWORK
TITLE =
      AN    "DB_Uscite".SbloccoFrenoAsseY;
      =     Q 41.1;
NETWORK
TITLE =
      A     "DB_Uscite".EV_ApriPortaRobot;
      =     Q 41.2;
NETWORK
TITLE =
      A     "DB_Uscite".EV_ChiudiPortaRobot;
      =     Q 41.3;
NETWORK
TITLE =
      A     "DB_Uscite".EvLubeAsseA;
      =     Q 42.0;
NETWORK
TITLE =
      A     "DB_Uscite".EvLubeAsseB;
      =     Q 42.1;
NETWORK
TITLE =
      A     "DB_Uscite".SoffieriaPezzo;
      =     Q 42.2;
NETWORK
TITLE =
      A     "DB_Uscite".PressurizzRettificaMola;
      =     Q 42.3;
NETWORK
TITLE =
      A     "DB_Uscite".PressurizzElettromandrin;
      =     Q 43.0;
NETWORK
TITLE =
      A     "DB_Uscite".Ev_SoffieriaPortapezzo;
      =     Q 43.1;
NETWORK
TITLE =
      A     "DB_Uscite".Ev_SoffieriaPortamola;
      =     Q 43.2;
NETWORK
TITLE =
      A     "DB_Uscite".EvGeneraleAriaON;
      =     Q 43.3;
END_FUNCTION

FUNCTION "FC Allarmi" : VOID	// FC 103
TITLE = FC Allarmi
AUTHOR : Asamec
VERSION : 0.1
VAR_TEMP
  Zero : BYTE ;
  RET_FILL : INT ;
END_VAR
BEGIN
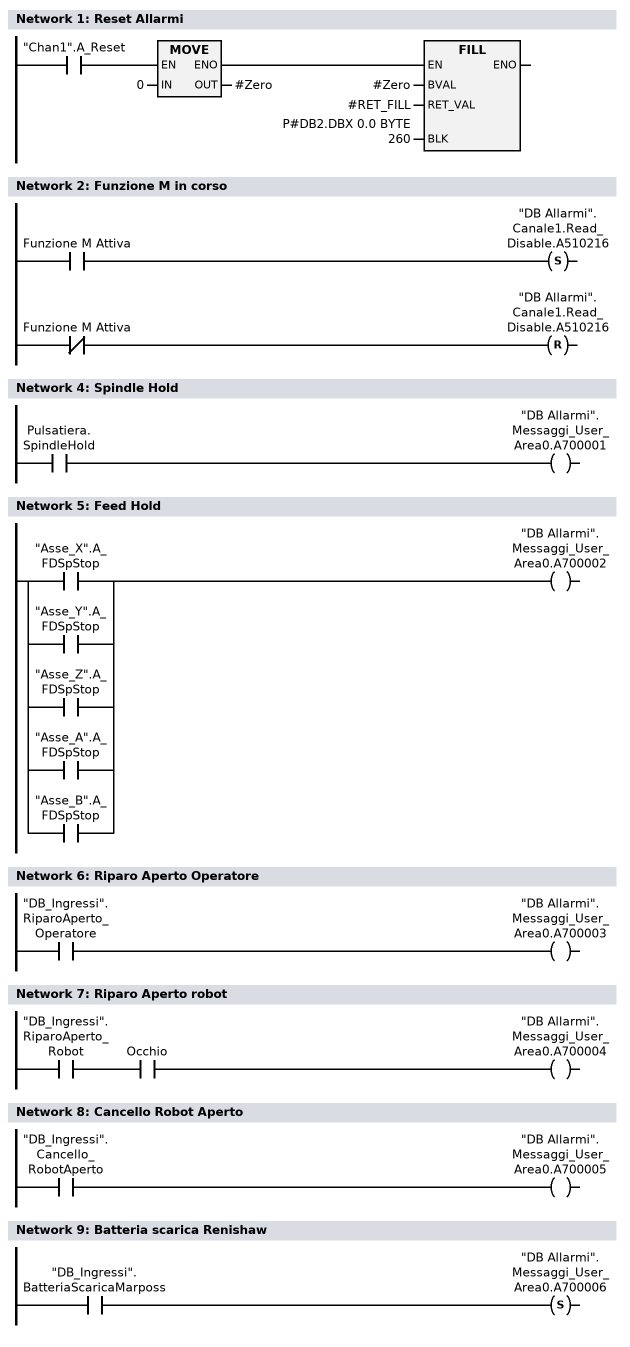
NETWORK
TITLE = Reset Allarmi
      A(;
      A     "Chan1".A_Reset;
      JNB   _001;
      L     0;
      T     #Zero;
      SET;
      SAVE;
      CLR;
_001: A     BR;
      );
      JNB   _002;
      CALL  "FILL" (
           BVAL                     := #Zero,
           RET_VAL                  := #RET_FILL,
           BLK                      := P#DB2.DBX 0.0 BYTE 260);
_002: NOP   0;
NETWORK
TITLE = Funzione M in corso
      A     "Funzione M Attiva";
      S     "DB Allarmi".Canale1.Read_Disable.A510216;
      AN    "Funzione M Attiva";
      R     "DB Allarmi".Canale1.Read_Disable.A510216;
      NOP   0;
NETWORK
TITLE = Messaggi
NETWORK
TITLE = Spindle Hold
      A     "Pulsatiera.SpindleHold";
      =     "DB Allarmi".Messaggi_User_Area0.A700001;
NETWORK
TITLE = Feed Hold
      O     "Asse_X".A_FDSpStop;
      O     "Asse_Y".A_FDSpStop;
      O     "Asse_Z".A_FDSpStop;
      O     "Asse_A".A_FDSpStop;
      O     "Asse_B".A_FDSpStop;
      =     "DB Allarmi".Messaggi_User_Area0.A700002;
NETWORK
TITLE = Riparo Aperto Operatore
      A     "DB_Ingressi".RiparoAperto_Operatore;
      =     "DB Allarmi".Messaggi_User_Area0.A700003;
NETWORK
TITLE = Riparo Aperto robot
      A     "DB_Ingressi".RiparoAperto_Robot;
      A     "Occhio";
      =     "DB Allarmi".Messaggi_User_Area0.A700004;
NETWORK
TITLE = Cancello Robot Aperto
      A     "DB_Ingressi".Cancello_RobotAperto;
      =     "DB Allarmi".Messaggi_User_Area0.A700005;
NETWORK
TITLE = Batteria scarica Renishaw
      A     "DB_Ingressi".BatteriaScaricaMarposs;
      S     "DB Allarmi".Messaggi_User_Area0.A700006;
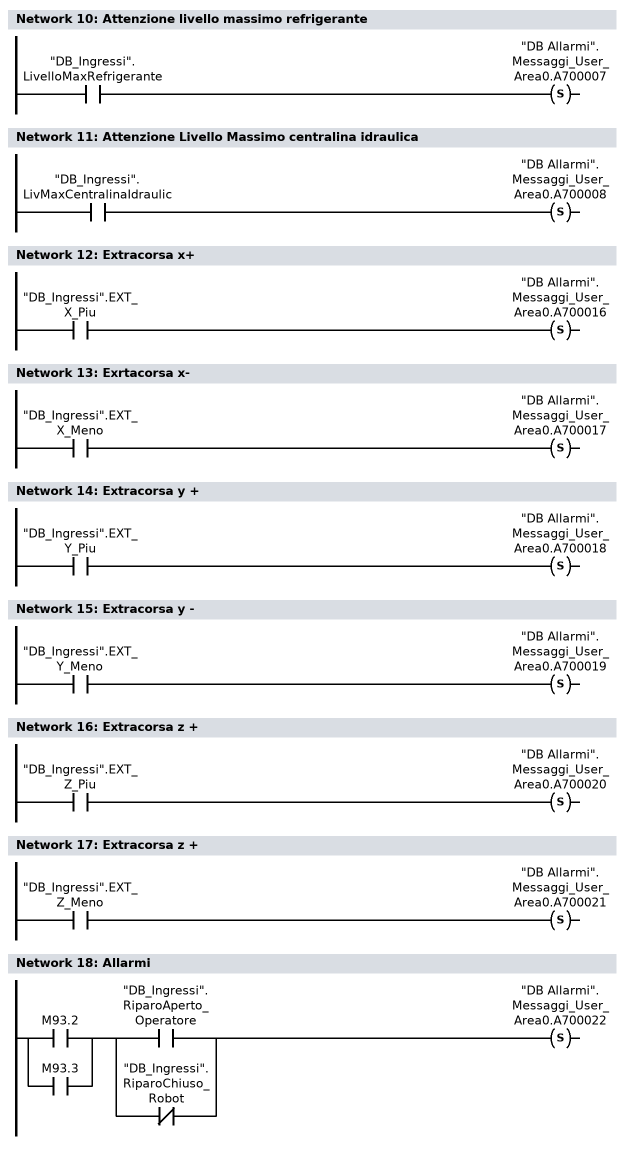
NETWORK
TITLE = Attenzione livello massimo refrigerante
      A     "DB_Ingressi".LivelloMaxRefrigerante;
      S     "DB Allarmi".Messaggi_User_Area0.A700007;
NETWORK
TITLE = Attenzione Livello Massimo centralina idraulica
      A     "DB_Ingressi".LivMaxCentralinaIdraulic;
      S     "DB Allarmi".Messaggi_User_Area0.A700008;
NETWORK
TITLE = Extracorsa x+
      A     "DB_Ingressi".EXT_X_Piu;
      S     "DB Allarmi".Messaggi_User_Area0.A700016;
NETWORK
TITLE = Exrtacorsa x-
      A     "DB_Ingressi".EXT_X_Meno;
      S     "DB Allarmi".Messaggi_User_Area0.A700017;
NETWORK
TITLE = Extracorsa y +
      A     "DB_Ingressi".EXT_Y_Piu;
      S     "DB Allarmi".Messaggi_User_Area0.A700018;
NETWORK
TITLE = Extracorsa y -
      A     "DB_Ingressi".EXT_Y_Meno;
      S     "DB Allarmi".Messaggi_User_Area0.A700019;
NETWORK
TITLE = Extracorsa z +
      A     "DB_Ingressi".EXT_Z_Piu;
      S     "DB Allarmi".Messaggi_User_Area0.A700020;
NETWORK
TITLE = Extracorsa z +
      A     "DB_Ingressi".EXT_Z_Meno;
      S     "DB Allarmi".Messaggi_User_Area0.A700021;
NETWORK
TITLE = Allarmi
      A(;
      O     "M93.2";
      O     "M93.3";
      );
      A(;
      O     "DB_Ingressi".RiparoAperto_Operatore;
      ON    "DB_Ingressi".RiparoChiuso_Robot;
      );
      S     "DB Allarmi".Messaggi_User_Area0.A700022;
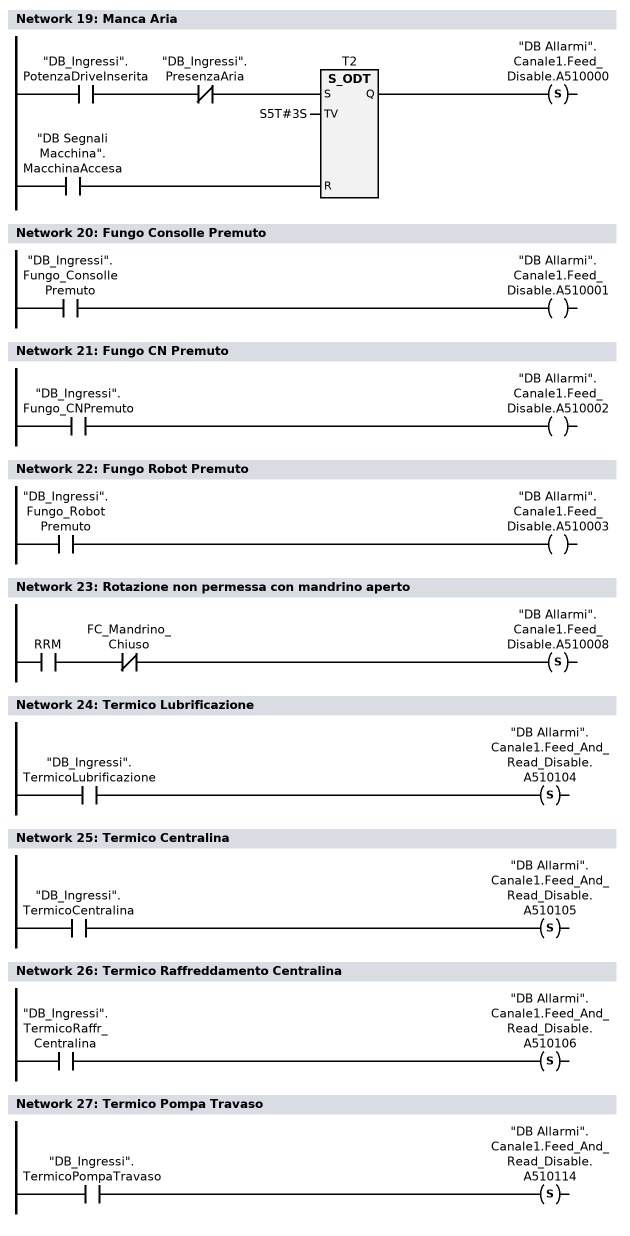
NETWORK
TITLE = Manca Aria
      A     "DB_Ingressi".PotenzaDriveInserita;
      AN    "DB_Ingressi".PresenzaAria;
      L     S5T#3S;
      SD    "T2";
      A     "DB Segnali Macchina".MacchinaAccesa;
      R     "T2";
      NOP   0;
      NOP   0;
      A     "T2";
      S     "DB Allarmi".Canale1.Feed_Disable.A510000;
NETWORK
TITLE = Fungo Consolle Premuto
      A     "DB_Ingressi".Fungo_ConsollePremuto;
      =     "DB Allarmi".Canale1.Feed_Disable.A510001;
NETWORK
TITLE = Fungo CN Premuto
      A     "DB_Ingressi".Fungo_CNPremuto;
      =     "DB Allarmi".Canale1.Feed_Disable.A510002;
NETWORK
TITLE = Fungo Robot Premuto
      A     "DB_Ingressi".Fungo_RobotPremuto;
      =     "DB Allarmi".Canale1.Feed_Disable.A510003;
NETWORK
TITLE = Rotazione non permessa con mandrino aperto
      A     "RRM";
      AN    "FC_Mandrino_Chiuso";
      S     "DB Allarmi".Canale1.Feed_Disable.A510008;
NETWORK
TITLE = Termico Lubrificazione
      A     "DB_Ingressi".TermicoLubrificazione;
      S     "DB Allarmi".Canale1.Feed_And_Read_Disable.A510104;
NETWORK
TITLE = Termico Centralina
      A     "DB_Ingressi".TermicoCentralina;
      S     "DB Allarmi".Canale1.Feed_And_Read_Disable.A510105;
NETWORK
TITLE = Termico Raffreddamento Centralina
      A     "DB_Ingressi".TermicoRaffr_Centralina;
      S     "DB Allarmi".Canale1.Feed_And_Read_Disable.A510106;
NETWORK
TITLE = Termico Pompa Travaso
      A     "DB_Ingressi".TermicoPompaTravaso;
      S     "DB Allarmi".Canale1.Feed_And_Read_Disable.A510114;
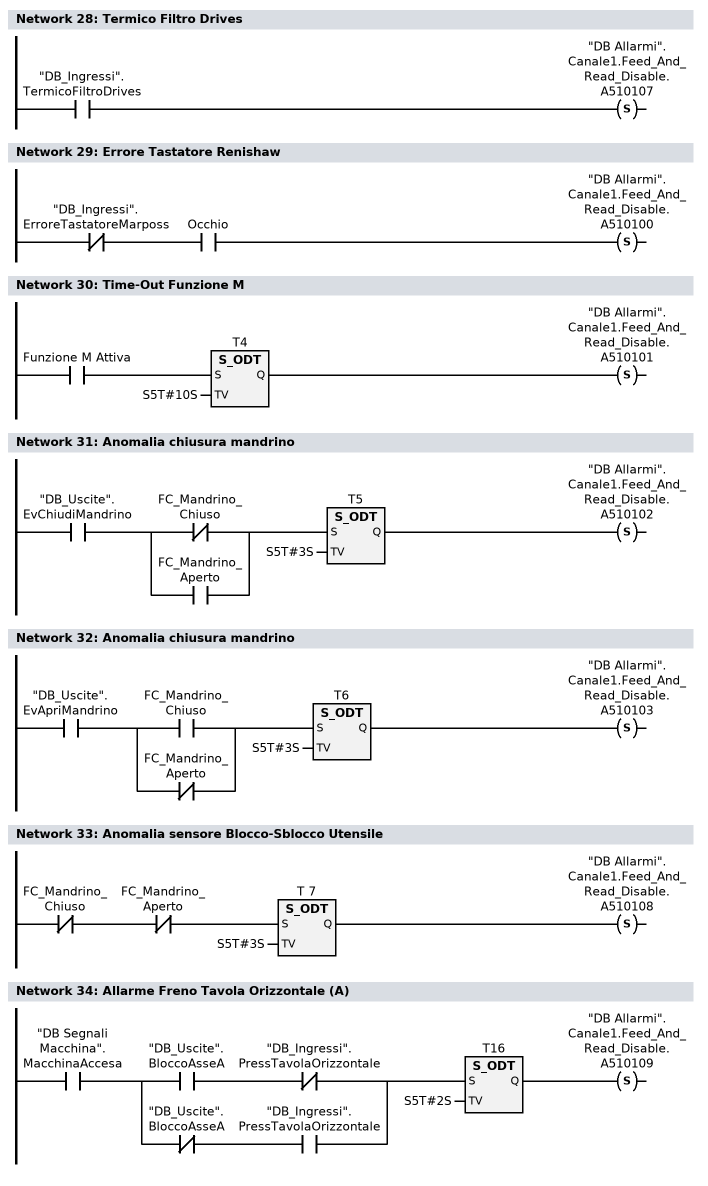
NETWORK
TITLE = Termico Filtro Drives
      A     "DB_Ingressi".TermicoFiltroDrives;
      S     "DB Allarmi".Canale1.Feed_And_Read_Disable.A510107;
NETWORK
TITLE = Errore Tastatore Renishaw
      AN    "DB_Ingressi".ErroreTastatoreMarposs;
      A     "Occhio";
      S     "DB Allarmi".Canale1.Feed_And_Read_Disable.A510100;
NETWORK
TITLE = Time-Out Funzione M
      A     "Funzione M Attiva";
      L     S5T#10S;
      SD    "T4";
      NOP   0;
      NOP   0;
      NOP   0;
      A     "T4";
      S     "DB Allarmi".Canale1.Feed_And_Read_Disable.A510101;
NETWORK
TITLE = Anomalia chiusura mandrino
      A     "DB_Uscite".EvChiudiMandrino;
      A(;
      ON    "FC_Mandrino_Chiuso";
      O     "FC_Mandrino_Aperto";
      );
      L     S5T#3S;
      SD    "T5";
      NOP   0;
      NOP   0;
      NOP   0;
      A     "T5";
      S     "DB Allarmi".Canale1.Feed_And_Read_Disable.A510102;
NETWORK
TITLE = Anomalia chiusura mandrino
      A     "DB_Uscite".EvApriMandrino;
      A(;
      O     "FC_Mandrino_Chiuso";
      ON    "FC_Mandrino_Aperto";
      );
      L     S5T#3S;
      SD    "T6";
      NOP   0;
      NOP   0;
      NOP   0;
      A     "T6";
      S     "DB Allarmi".Canale1.Feed_And_Read_Disable.A510103;
NETWORK
TITLE = Anomalia sensore Blocco-Sblocco Utensile
      AN    "FC_Mandrino_Chiuso";
      AN    "FC_Mandrino_Aperto";
      L     S5T#3S;
      SD    T 7;
      NOP   0;
      NOP   0;
      NOP   0;
      A     T 7;
      S     "DB Allarmi".Canale1.Feed_And_Read_Disable.A510108;
NETWORK
TITLE = Allarme Freno Tavola Orizzontale (A)
      A     "DB Segnali Macchina".MacchinaAccesa;
      A(;
      A     "DB_Uscite".BloccoAsseA;
      AN    "DB_Ingressi".PressTavolaOrizzontale;
      O;
      AN    "DB_Uscite".BloccoAsseA;
      A     "DB_Ingressi".PressTavolaOrizzontale;
      );
      L     S5T#2S;
      SD    "T16";
      NOP   0;
      NOP   0;
      NOP   0;
      A     "T16";
      S     "DB Allarmi".Canale1.Feed_And_Read_Disable.A510109;
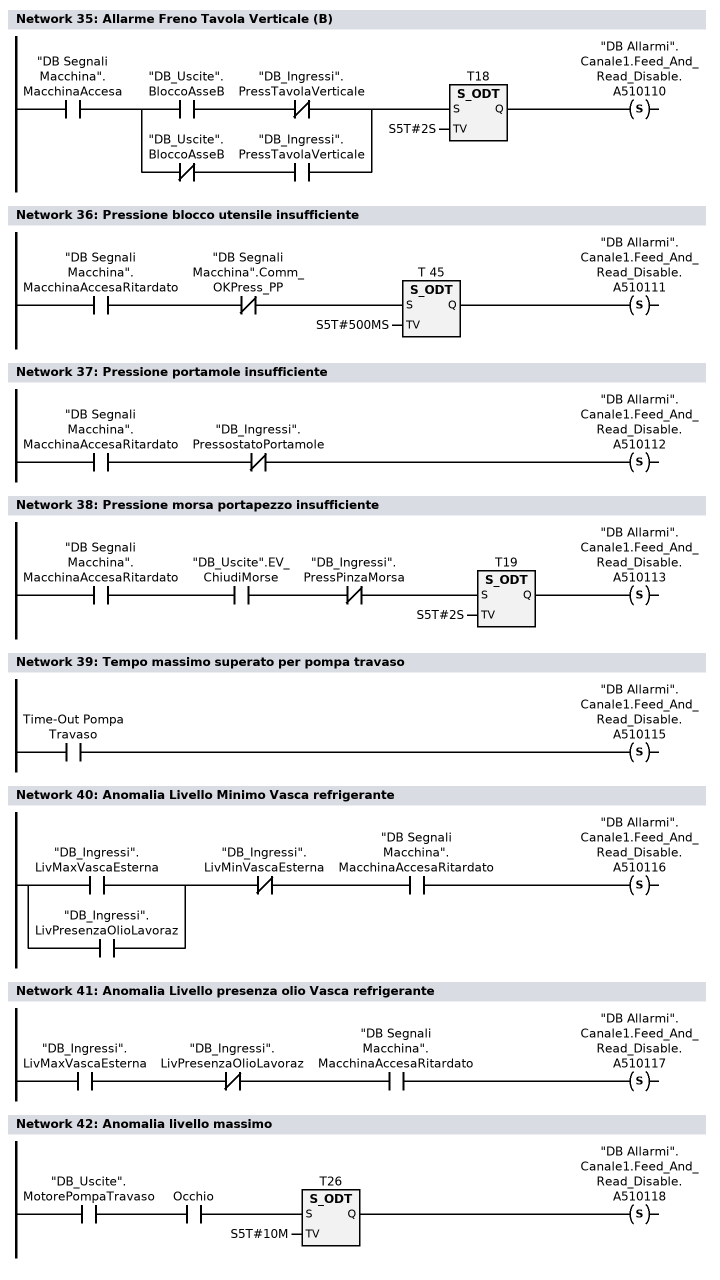
NETWORK
TITLE = Allarme Freno Tavola Verticale (B)
      A     "DB Segnali Macchina".MacchinaAccesa;
      A(;
      A     "DB_Uscite".BloccoAsseB;
      AN    "DB_Ingressi".PressTavolaVerticale;
      O;
      AN    "DB_Uscite".BloccoAsseB;
      A     "DB_Ingressi".PressTavolaVerticale;
      );
      L     S5T#2S;
      SD    "T18";
      NOP   0;
      NOP   0;
      NOP   0;
      A     "T18";
      S     "DB Allarmi".Canale1.Feed_And_Read_Disable.A510110;
NETWORK
TITLE = Pressione blocco utensile insufficiente
      A     "DB Segnali Macchina".MacchinaAccesaRitardato;
      AN    "DB Segnali Macchina".Comm_OKPress_PP;
      L     S5T#500MS;
      SD    T 45;
      NOP   0;
      NOP   0;
      NOP   0;
      A     T 45;
      S     "DB Allarmi".Canale1.Feed_And_Read_Disable.A510111;
NETWORK
TITLE = Pressione portamole insufficiente
      A     "DB Segnali Macchina".MacchinaAccesaRitardato;
      AN    "DB_Ingressi".PressostatoPortamole;
      S     "DB Allarmi".Canale1.Feed_And_Read_Disable.A510112;
NETWORK
TITLE = Pressione morsa portapezzo insufficiente
      A     "DB Segnali Macchina".MacchinaAccesaRitardato;
      A     "DB_Uscite".EV_ChiudiMorse;
      AN    "DB_Ingressi".PressPinzaMorsa;
      L     S5T#2S;
      SD    "T19";
      NOP   0;
      NOP   0;
      NOP   0;
      A     "T19";
      S     "DB Allarmi".Canale1.Feed_And_Read_Disable.A510113;
NETWORK
TITLE = Tempo massimo superato per pompa travaso
      A     "Time-Out Pompa Travaso";
      S     "DB Allarmi".Canale1.Feed_And_Read_Disable.A510115;
NETWORK
TITLE = Anomalia Livello Minimo Vasca refrigerante
      A(;
      O     "DB_Ingressi".LivMaxVascaEsterna;
      O     "DB_Ingressi".LivPresenzaOlioLavoraz;
      );
      AN    "DB_Ingressi".LivMinVascaEsterna;
      A     "DB Segnali Macchina".MacchinaAccesaRitardato;
      S     "DB Allarmi".Canale1.Feed_And_Read_Disable.A510116;
NETWORK
TITLE = Anomalia Livello presenza olio Vasca refrigerante
      A     "DB_Ingressi".LivMaxVascaEsterna;
      AN    "DB_Ingressi".LivPresenzaOlioLavoraz;
      A     "DB Segnali Macchina".MacchinaAccesaRitardato;
      S     "DB Allarmi".Canale1.Feed_And_Read_Disable.A510117;
NETWORK
TITLE = Anomalia livello massimo
      A     "DB_Uscite".MotorePompaTravaso;
      A     "Occhio";
      L     S5T#10M;
      SD    "T26";
      NOP   0;
      NOP   0;
      NOP   0;
      A     "T26";
      S     "DB Allarmi".Canale1.Feed_And_Read_Disable.A510118;
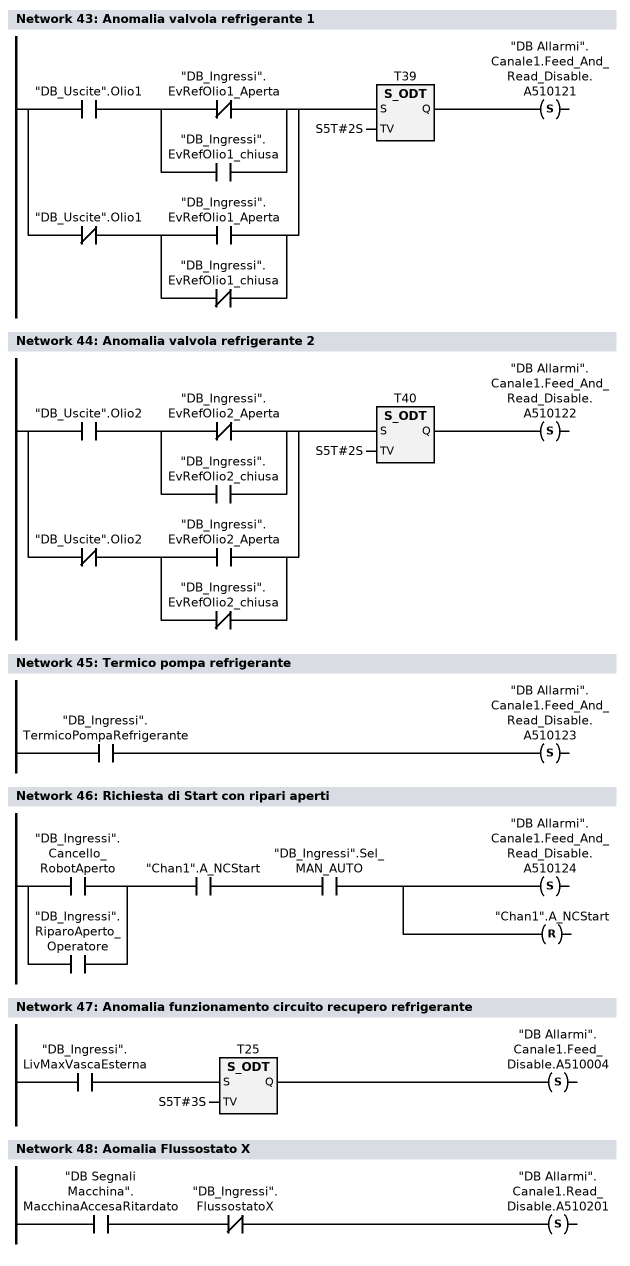
NETWORK
TITLE = Anomalia valvola refrigerante 1
      A(;
      A     "DB_Uscite".Olio1;
      A(;
      ON    "DB_Ingressi".EvRefOlio1_Aperta;
      O     "DB_Ingressi".EvRefOlio1_chiusa;
      );
      O;
      AN    "DB_Uscite".Olio1;
      A(;
      O     "DB_Ingressi".EvRefOlio1_Aperta;
      ON    "DB_Ingressi".EvRefOlio1_chiusa;
      );
      );
      L     S5T#2S;
      SD    "T39";
      NOP   0;
      NOP   0;
      NOP   0;
      A     "T39";
      S     "DB Allarmi".Canale1.Feed_And_Read_Disable.A510121;
NETWORK
TITLE = Anomalia valvola refrigerante 2
      A(;
      A     "DB_Uscite".Olio2;
      A(;
      ON    "DB_Ingressi".EvRefOlio2_Aperta;
      O     "DB_Ingressi".EvRefOlio2_chiusa;
      );
      O;
      AN    "DB_Uscite".Olio2;
      A(;
      O     "DB_Ingressi".EvRefOlio2_Aperta;
      ON    "DB_Ingressi".EvRefOlio2_chiusa;
      );
      );
      L     S5T#2S;
      SD    "T40";
      NOP   0;
      NOP   0;
      NOP   0;
      A     "T40";
      S     "DB Allarmi".Canale1.Feed_And_Read_Disable.A510122;
NETWORK
TITLE = Termico pompa refrigerante
      A     "DB_Ingressi".TermicoPompaRefrigerante;
      S     "DB Allarmi".Canale1.Feed_And_Read_Disable.A510123;
NETWORK
TITLE = Richiesta di Start con ripari aperti
      A(;
      O     "DB_Ingressi".Cancello_RobotAperto;
      O     "DB_Ingressi".RiparoAperto_Operatore;
      );
      A     "Chan1".A_NCStart;
      A     "DB_Ingressi".Sel_MAN_AUTO;
      S     "DB Allarmi".Canale1.Feed_And_Read_Disable.A510124;
      R     "Chan1".A_NCStart;
NETWORK
TITLE = Anomalia funzionamento circuito recupero refrigerante
      A     "DB_Ingressi".LivMaxVascaEsterna;
      L     S5T#3S;
      SD    "T25";
      NOP   0;
      NOP   0;
      NOP   0;
      A     "T25";
      S     "DB Allarmi".Canale1.Feed_Disable.A510004;
NETWORK
TITLE = Aomalia Flussostato X
      A     "DB Segnali Macchina".MacchinaAccesaRitardato;
      AN    "DB_Ingressi".FlussostatoX;
      S     "DB Allarmi".Canale1.Read_Disable.A510201;
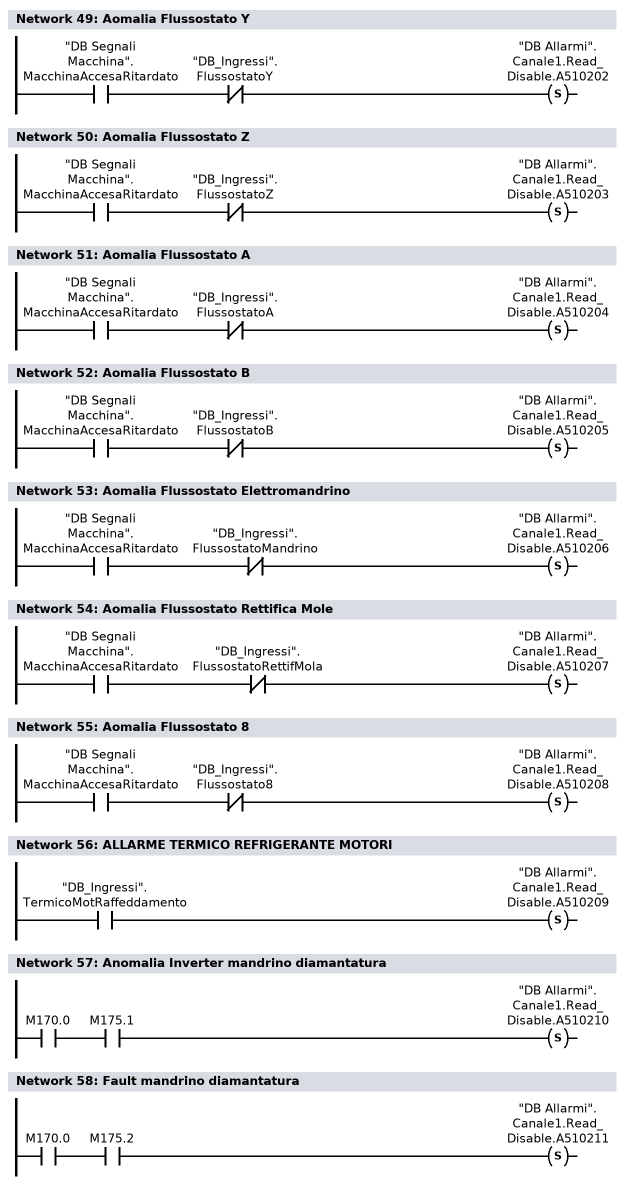
NETWORK
TITLE = Aomalia Flussostato Y
      A     "DB Segnali Macchina".MacchinaAccesaRitardato;
      AN    "DB_Ingressi".FlussostatoY;
      S     "DB Allarmi".Canale1.Read_Disable.A510202;
NETWORK
TITLE = Aomalia Flussostato Z
      A     "DB Segnali Macchina".MacchinaAccesaRitardato;
      AN    "DB_Ingressi".FlussostatoZ;
      S     "DB Allarmi".Canale1.Read_Disable.A510203;
NETWORK
TITLE = Aomalia Flussostato A
      A     "DB Segnali Macchina".MacchinaAccesaRitardato;
      AN    "DB_Ingressi".FlussostatoA;
      S     "DB Allarmi".Canale1.Read_Disable.A510204;
NETWORK
TITLE = Aomalia Flussostato B
      A     "DB Segnali Macchina".MacchinaAccesaRitardato;
      AN    "DB_Ingressi".FlussostatoB;
      S     "DB Allarmi".Canale1.Read_Disable.A510205;
NETWORK
TITLE = Aomalia Flussostato Elettromandrino
      A     "DB Segnali Macchina".MacchinaAccesaRitardato;
      AN    "DB_Ingressi".FlussostatoMandrino;
      S     "DB Allarmi".Canale1.Read_Disable.A510206;
NETWORK
TITLE = Aomalia Flussostato Rettifica Mole
      A     "DB Segnali Macchina".MacchinaAccesaRitardato;
      AN    "DB_Ingressi".FlussostatoRettifMola;
      S     "DB Allarmi".Canale1.Read_Disable.A510207;
NETWORK
TITLE = Aomalia Flussostato 8
      A     "DB Segnali Macchina".MacchinaAccesaRitardato;
      AN    "DB_Ingressi".Flussostato8;
      S     "DB Allarmi".Canale1.Read_Disable.A510208;
NETWORK
TITLE = ALLARME TERMICO REFRIGERANTE MOTORI
      A     "DB_Ingressi".TermicoMotRaffeddamento;
      S     "DB Allarmi".Canale1.Read_Disable.A510209;
NETWORK
TITLE = Anomalia Inverter mandrino diamantatura
      A     "M170.0";
      A     "M175.1";
      S     "DB Allarmi".Canale1.Read_Disable.A510210;
NETWORK
TITLE = Fault mandrino diamantatura
      A     "M170.0";
      A     "M175.2";
      S     "DB Allarmi".Canale1.Read_Disable.A510211;
END_FUNCTION

FUNCTION "FC Sicurezze" : VOID	// FC 104
TITLE = Gestione sicurezze macchina
AUTHOR : Asamec
VERSION : 0.1
BEGIN
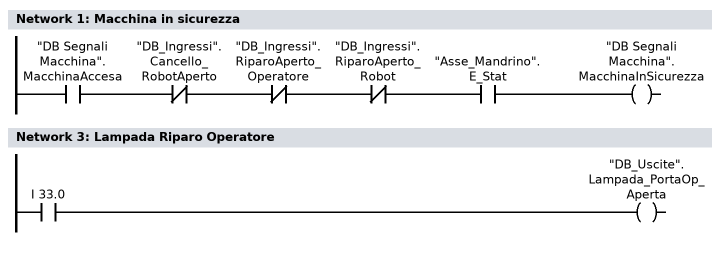
NETWORK
TITLE = Macchina in sicurezza
      A     "DB Segnali Macchina".MacchinaAccesa;
      AN    "DB_Ingressi".Cancello_RobotAperto;
      AN    "DB_Ingressi".RiparoAperto_Operatore;
      AN    "DB_Ingressi".RiparoAperto_Robot;
      A     "Asse_Mandrino".E_Stat;
      =     "DB Segnali Macchina".MacchinaInSicurezza;
NETWORK
TITLE = Sblocco Riparo Operatore
      A     I 6.1;
      O     I 42.0;
      AN    "BAG".E_AUTO;
      A(;
      A     "Chan1".E_ChanReset;
      ON    "DB Segnali Macchina".MacchinaAccesa;
      );
      FP    "M92.0";
      X     "M92.1";
      =     "M92.1";
      =     Q 4.1;
NETWORK
TITLE = Lampada Riparo Operatore
      A     I 33.0;
      =     "DB_Uscite".Lampada_PortaOp_Aperta;
END_FUNCTION

FUNCTION "FC Mandrino" : VOID	// FC 105
AUTHOR : Asamec
VERSION : 0.1
BEGIN
